REGION Network 10: Temperature Reached Conditions
   RUNG wire#powerrail
      Contact( #Selected )
      Contact( #Running )
      Contact( #Started )
      wire#w1
      { S7_Templates := "SrcType := Int" } EQ_Contact(in1 := #TemperatureControlSel, in2 := 0)
      wire#w2
      { S7_Templates := "SrcType := Real" } GE_Contact(in1 := #ActualTemperature, in2 := #SetTemperature)
      S_Coil( #HeatTempReached )
   END_RUNG
   RUNG wire#w2
      { S7_Templates := "SrcType := Real" } LE_Contact(in1 := #ActualTemperature, in2 := #TemperatureTolNeg)
      R_Coil( #HeatTempReached )
   END_RUNG
   RUNG wire#w1
      { S7_Templates := "SrcType := Int" } EQ_Contact(in1 := #TemperatureControlSel, in2 := 1)
      wire#w3
      { S7_Templates := "SrcType := Real" } LE_Contact(in1 := #ActualTemperature, in2 := #SetTemperature)
      S_Coil( #CoolTempReached )
   END_RUNG
   RUNG wire#w3
      { S7_Templates := "SrcType := Real" } GE_Contact(in1 := #ActualTemperature, in2 := #TemperatureTolPos)
      R_Coil( #CoolTempReached )
   END_RUNG
   // the same network as SCL:
   #_w1 := #Selected AND #Running AND #Started;
   #_w2 := #_w1 AND (#TemperatureControlSel = 0);
   IF #_w2 AND (#ActualTemperature >= #SetTemperature) THEN #HeatTempReached := TRUE; END_IF;
   IF #_w2 AND (#ActualTemperature <= #TemperatureTolNeg) THEN #HeatTempReached := FALSE; END_IF;
   #_w3 := #_w1 AND (#TemperatureControlSel = 1);
   IF #_w3 AND (#ActualTemperature <= #SetTemperature) THEN #CoolTempReached := TRUE; END_IF;
   IF #_w3 AND (#ActualTemperature >= #TemperatureTolPos) THEN #CoolTempReached := FALSE; END_IF;
END_REGION

REGION Network 11: Timer
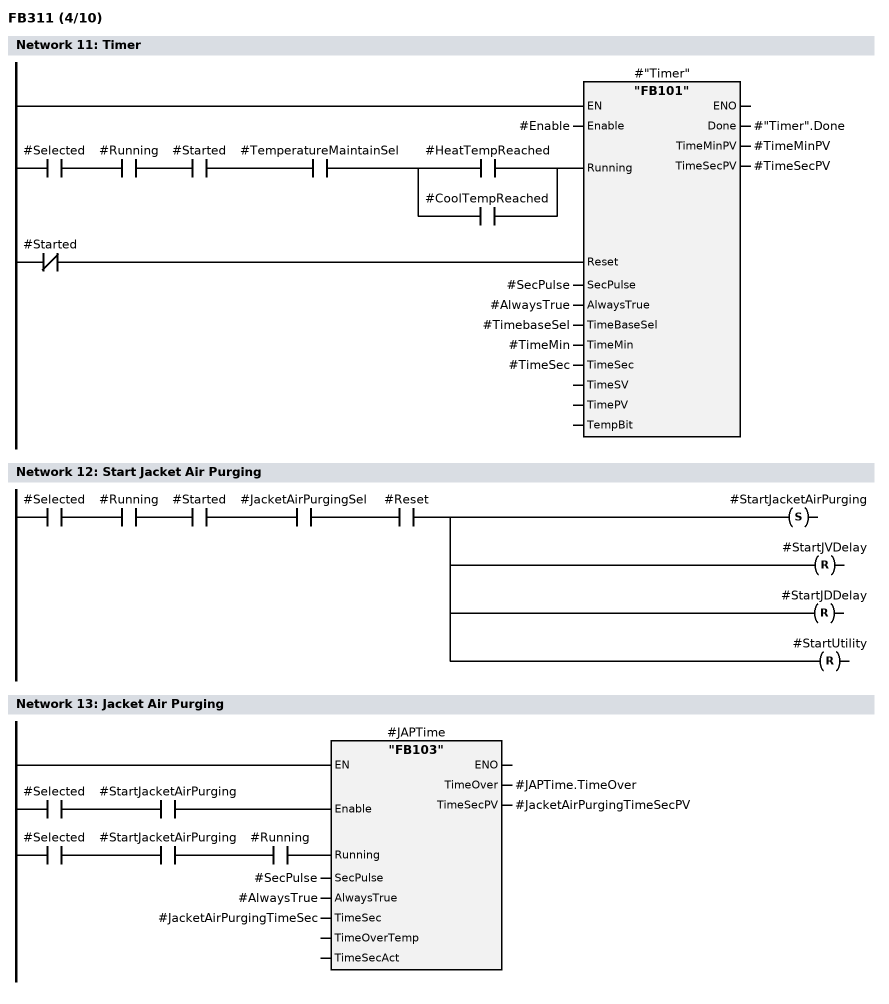
   RUNG wire#powerrail
      #"Timer"(Running := wire#w2, Reset := wire#w3, Enable := #Enable, SecPulse := #SecPulse, AlwaysTrue := #AlwaysTrue, TimeBaseSel := #TimebaseSel, TimeMin := #TimeMin, TimeSec := #TimeSec, TimeSV :=, TimePV :=, TempBit :=, Done => #"Timer".Done, TimeMinPV => #TimeMinPV, TimeSecPV => #TimeSecPV)
   END_RUNG
   RUNG wire#powerrail
      Contact( #Selected )
      Contact( #Running )
      Contact( #Started )
      Contact( #TemperatureMaintainSel )
      wire#w1
      Contact( #HeatTempReached )
   END_RUNG wire#w2
   RUNG wire#w1
      Contact( #CoolTempReached )
   END_RUNG wire#w2
   RUNG wire#powerrail
      I_Contact( #Started )
   END_RUNG wire#w3
   // the same network as SCL:
   #"Timer"(Enable := #Enable,   // "FB101"
            Running := #Selected AND #Running AND #Started AND #TemperatureMaintainSel AND (#HeatTempReached OR #CoolTempReached),
            Reset := NOT #Started,
            SecPulse := #SecPulse,
            AlwaysTrue := #AlwaysTrue,
            TimeBaseSel := #TimebaseSel,
            TimeMin := #TimeMin,
            TimeSec := #TimeSec,
            Done => #"Timer".Done,
            TimeMinPV => #TimeMinPV,
            TimeSecPV => #TimeSecPV);
END_REGION

REGION Network 12: Start Jacket Air Purging
   RUNG wire#powerrail
      Contact( #Selected )
      Contact( #Running )
      Contact( #Started )
      Contact( #JacketAirPurgingSel )
      Contact( #Reset )
      wire#w1
      S_Coil( #StartJacketAirPurging )
   END_RUNG
   RUNG wire#w1
      R_Coil( #StartJVDelay )
   END_RUNG
   RUNG wire#w1
      R_Coil( #StartJDDelay )
   END_RUNG
   RUNG wire#w1
      R_Coil( #StartUtility )
   END_RUNG
   // the same network as SCL:
   IF #Selected AND #Running AND #Started AND #JacketAirPurgingSel AND #Reset THEN
       #StartJacketAirPurging := TRUE;
       #StartJVDelay := FALSE;
       #StartJDDelay := FALSE;
       #StartUtility := FALSE;
   END_IF;
END_REGION

REGION Network 13: Jacket Air Purging
   RUNG wire#powerrail
      #JAPTime(Enable := wire#w1, Running := wire#w2, SecPulse := #SecPulse, AlwaysTrue := #AlwaysTrue, TimeSec := #JacketAirPurgingTimeSec, TimeOverTemp :=, TimeSecAct :=, TimeOver => #JAPTime.TimeOver, TimeSecPV => #JacketAirPurgingTimeSecPV)
   END_RUNG
   RUNG wire#powerrail
      Contact( #Selected )
      Contact( #StartJacketAirPurging )
   END_RUNG wire#w1
   RUNG wire#powerrail
      Contact( #Selected )
      Contact( #StartJacketAirPurging )
      Contact( #Running )
   END_RUNG wire#w2
   // the same network as SCL:
   #JAPTime(Enable := #Selected AND #StartJacketAirPurging,   // "FB103"
            Running := #Selected AND #StartJacketAirPurging AND #Running,
            SecPulse := #SecPulse,
            AlwaysTrue := #AlwaysTrue,
            TimeSec := #JacketAirPurgingTimeSec,
            TimeOver => #JAPTime.TimeOver,
            TimeSecPV => #JacketAirPurgingTimeSecPV);
END_REGION

REGION Network 14: Over
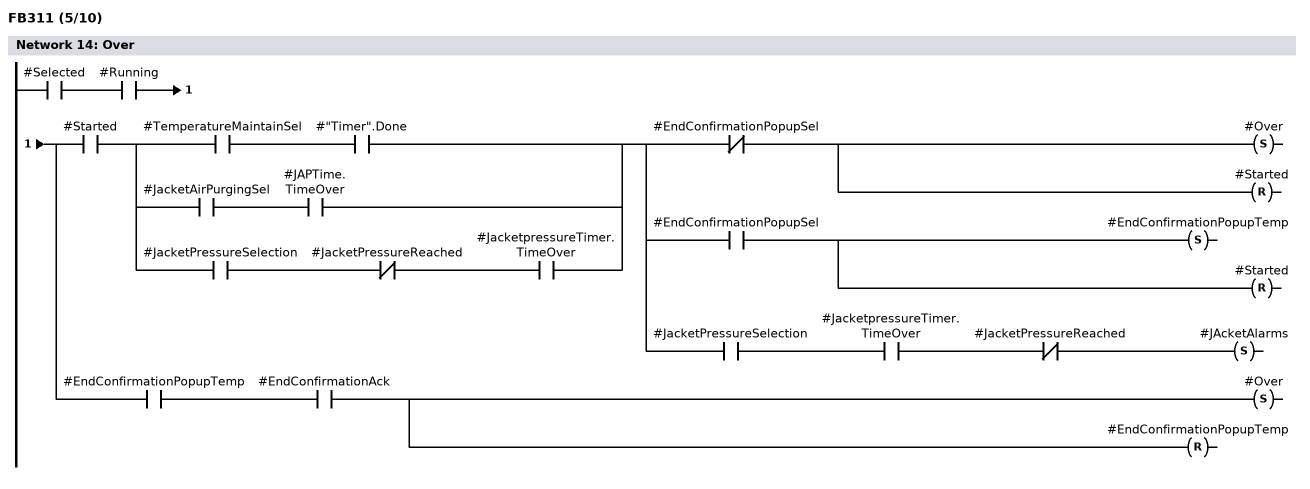
   RUNG wire#powerrail
      Contact( #Selected )
      Contact( #Running )
      wire#w1
      Contact( #Started )
      wire#w2
      Contact( #TemperatureMaintainSel )
      Contact( #"Timer".Done )
      wire#w3
      I_Contact( #EndConfirmationPopupSel )
      wire#w4
      S_Coil( #Over )
   END_RUNG
   RUNG wire#w2
      Contact( #JacketAirPurgingSel )
      Contact( #JAPTime.TimeOver )
   END_RUNG wire#w3
   RUNG wire#w2
      Contact( #JacketPressureSelection )
      I_Contact( #JacketPressureReached )
      Contact( #JacketpressureTimer.TimeOver )
   END_RUNG wire#w3
   RUNG wire#w4
      R_Coil( #Started )
   END_RUNG
   RUNG wire#w3
      Contact( #EndConfirmationPopupSel )
      wire#w5
      S_Coil( #EndConfirmationPopupTemp )
   END_RUNG
   RUNG wire#w5
      R_Coil( #Started )
   END_RUNG
   RUNG wire#w3
      Contact( #JacketPressureSelection )
      Contact( #JacketpressureTimer.TimeOver )
      I_Contact( #JacketPressureReached )
      S_Coil( #JAcketAlarms )
   END_RUNG
   RUNG wire#w1
      Contact( #EndConfirmationPopupTemp )
      Contact( #EndConfirmationAck )
      wire#w6
      S_Coil( #Over )
   END_RUNG
   RUNG wire#w6
      R_Coil( #EndConfirmationPopupTemp )
   END_RUNG
   // the same network as SCL:
   #_w1 := #Selected AND #Running;
   #_w2 := #_w1 AND #Started AND ((#TemperatureMaintainSel AND #"Timer".Done) OR (#JacketAirPurgingSel AND #JAPTime.TimeOver) OR (#JacketPressureSelection AND NOT #JacketPressureReached AND #JacketpressureTimer.TimeOver));
   IF #_w2 AND NOT #EndConfirmationPopupSel THEN
       #Over := TRUE;
       #Started := FALSE;
   END_IF;
   IF #_w2 AND #EndConfirmationPopupSel THEN
       #EndConfirmationPopupTemp := TRUE;
       #Started := FALSE;
   END_IF;
   IF #_w2 AND #JacketPressureSelection AND #JacketpressureTimer.TimeOver AND NOT #JacketPressureReached THEN
       #JAcketAlarms := TRUE;
   END_IF;
   IF #_w1 AND #EndConfirmationPopupTemp AND #EndConfirmationAck THEN
       #Over := TRUE;
       #EndConfirmationPopupTemp := FALSE;
   END_IF;
END_REGION

REGION Network 15: Outputs
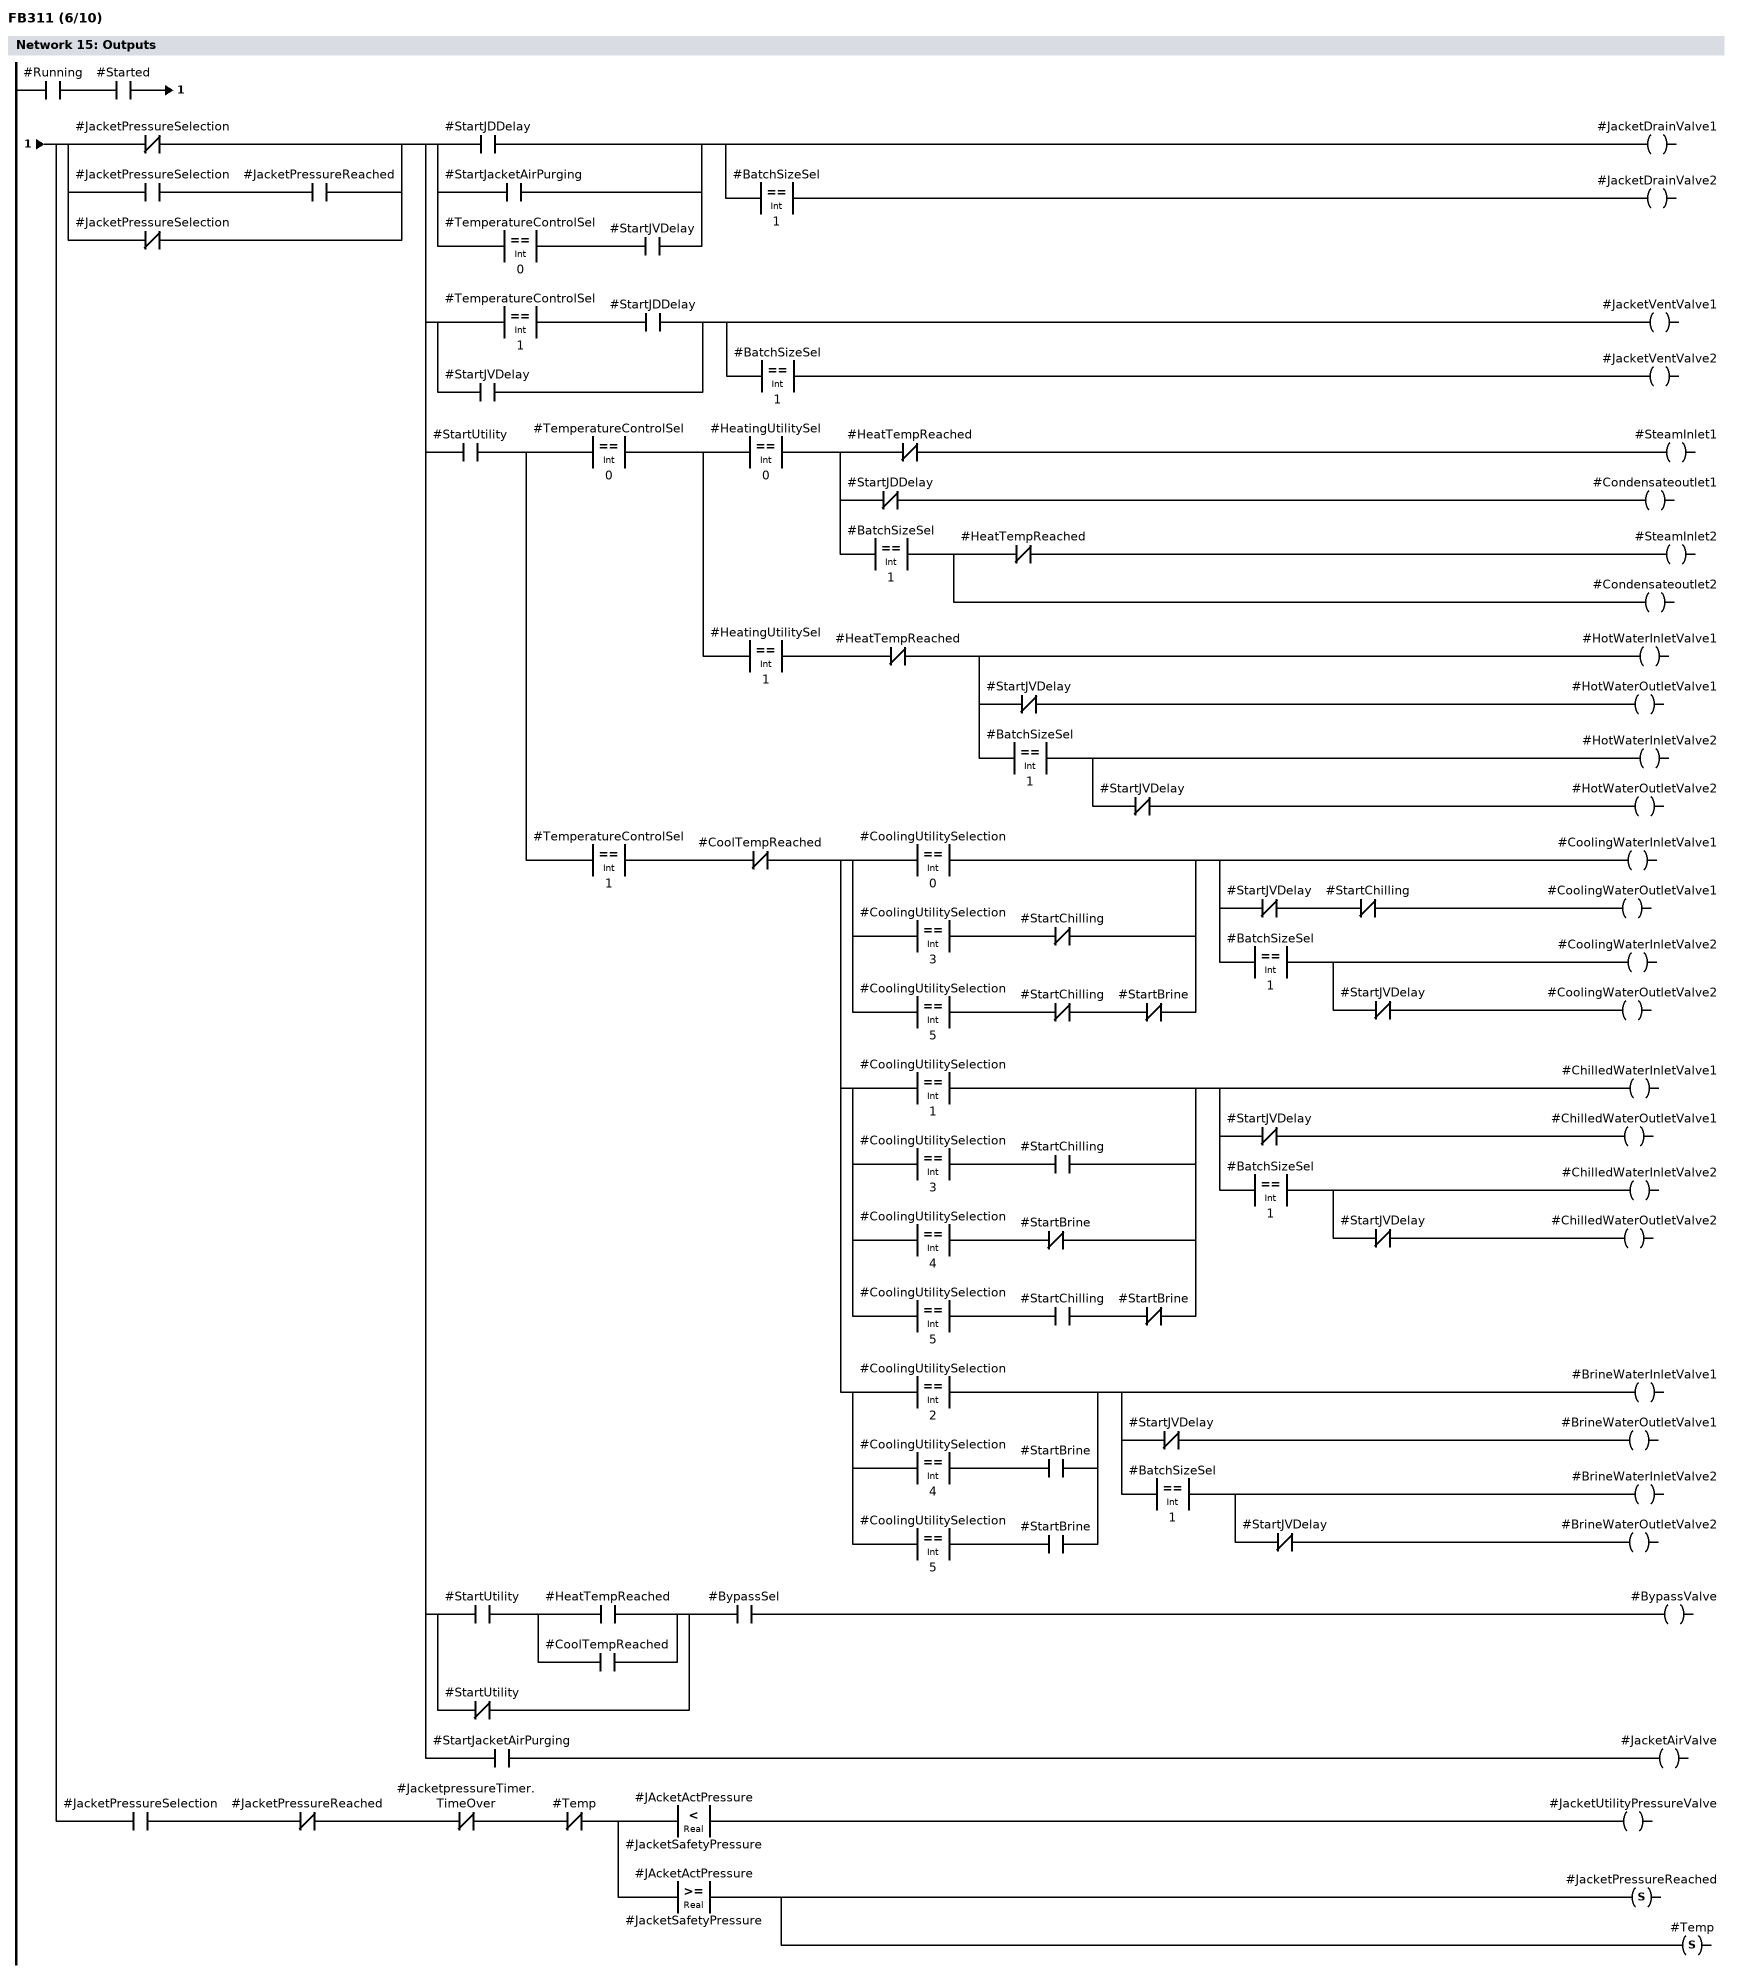
   RUNG wire#powerrail
      Contact( #Running )
      Contact( #Started )
      wire#w1
      I_Contact( #JacketPressureSelection )
      wire#w2
      Contact( #StartJDDelay )
      wire#w3
      Coil( #JacketDrainValve1 )
   END_RUNG
   RUNG wire#w1
      Contact( #JacketPressureSelection )
      Contact( #JacketPressureReached )
   END_RUNG wire#w2
   RUNG wire#w1
      I_Contact( #JacketPressureSelection )
   END_RUNG wire#w2
   RUNG wire#w2
      Contact( #StartJacketAirPurging )
   END_RUNG wire#w3
   RUNG wire#w2
      { S7_Templates := "SrcType := Int" } EQ_Contact(in1 := #TemperatureControlSel, in2 := 0)
      Contact( #StartJVDelay )
   END_RUNG wire#w3
   RUNG wire#w3
      { S7_Templates := "SrcType := Int" } EQ_Contact(in1 := #BatchSizeSel, in2 := 1)
      Coil( #JacketDrainValve2 )
   END_RUNG
   RUNG wire#w2
      { S7_Templates := "SrcType := Int" } EQ_Contact(in1 := #TemperatureControlSel, in2 := 1)
      Contact( #StartJDDelay )
      wire#w4
      Coil( #JacketVentValve1 )
   END_RUNG
   RUNG wire#w2
      Contact( #StartJVDelay )
   END_RUNG wire#w4
   RUNG wire#w4
      { S7_Templates := "SrcType := Int" } EQ_Contact(in1 := #BatchSizeSel, in2 := 1)
      Coil( #JacketVentValve2 )
   END_RUNG
   RUNG wire#w2
      Contact( #StartUtility )
      wire#w5
      { S7_Templates := "SrcType := Int" } EQ_Contact(in1 := #TemperatureControlSel, in2 := 0)
      wire#w6
      { S7_Templates := "SrcType := Int" } EQ_Contact(in1 := #HeatingUtilitySel, in2 := 0)
      wire#w7
      I_Contact( #HeatTempReached )
      Coil( #SteamInlet1 )
   END_RUNG
   RUNG wire#w7
      I_Contact( #StartJDDelay )
      Coil( #Condensateoutlet1 )
   END_RUNG
   RUNG wire#w7
      { S7_Templates := "SrcType := Int" } EQ_Contact(in1 := #BatchSizeSel, in2 := 1)
      wire#w8
      I_Contact( #HeatTempReached )
      Coil( #SteamInlet2 )
   END_RUNG
   RUNG wire#w8
      Coil( #Condensateoutlet2 )
   END_RUNG
   RUNG wire#w6
      { S7_Templates := "SrcType := Int" } EQ_Contact(in1 := #HeatingUtilitySel, in2 := 1)
      I_Contact( #HeatTempReached )
      wire#w9
      Coil( #HotWaterInletValve1 )
   END_RUNG
   RUNG wire#w9
      I_Contact( #StartJVDelay )
      Coil( #HotWaterOutletValve1 )
   END_RUNG
   RUNG wire#w9
      { S7_Templates := "SrcType := Int" } EQ_Contact(in1 := #BatchSizeSel, in2 := 1)
      wire#w10
      Coil( #HotWaterInletValve2 )
   END_RUNG
   RUNG wire#w10
      I_Contact( #StartJVDelay )
      Coil( #HotWaterOutletValve2 )
   END_RUNG
   RUNG wire#w5
      { S7_Templates := "SrcType := Int" } EQ_Contact(in1 := #TemperatureControlSel, in2 := 1)
      I_Contact( #CoolTempReached )
      wire#w11
      { S7_Templates := "SrcType := Int" } EQ_Contact(in1 := #CoolingUtilitySelection, in2 := 0)
      wire#w12
      Coil( #CoolingWaterInletValve1 )
   END_RUNG
   RUNG wire#w11
      { S7_Templates := "SrcType := Int" } EQ_Contact(in1 := #CoolingUtilitySelection, in2 := 3)
      I_Contact( #StartChilling )
   END_RUNG wire#w12
   RUNG wire#w11
      { S7_Templates := "SrcType := Int" } EQ_Contact(in1 := #CoolingUtilitySelection, in2 := 5)
      I_Contact( #StartChilling )
      I_Contact( #StartBrine )
   END_RUNG wire#w12
   RUNG wire#w12
      I_Contact( #StartJVDelay )
      I_Contact( #StartChilling )
      Coil( #CoolingWaterOutletValve1 )
   END_RUNG
   RUNG wire#w12
      { S7_Templates := "SrcType := Int" } EQ_Contact(in1 := #BatchSizeSel, in2 := 1)
      wire#w13
      Coil( #CoolingWaterInletValve2 )
   END_RUNG
   RUNG wire#w13
      I_Contact( #StartJVDelay )
      Coil( #CoolingWaterOutletValve2 )
   END_RUNG
   RUNG wire#w11
      { S7_Templates := "SrcType := Int" } EQ_Contact(in1 := #CoolingUtilitySelection, in2 := 1)
      wire#w14
      Coil( #ChilledWaterInletValve1 )
   END_RUNG
   RUNG wire#w11
      { S7_Templates := "SrcType := Int" } EQ_Contact(in1 := #CoolingUtilitySelection, in2 := 3)
      Contact( #StartChilling )
   END_RUNG wire#w14
   RUNG wire#w11
      { S7_Templates := "SrcType := Int" } EQ_Contact(in1 := #CoolingUtilitySelection, in2 := 4)
      I_Contact( #StartBrine )
   END_RUNG wire#w14
   RUNG wire#w11
      { S7_Templates := "SrcType := Int" } EQ_Contact(in1 := #CoolingUtilitySelection, in2 := 5)
      Contact( #StartChilling )
      I_Contact( #StartBrine )
   END_RUNG wire#w14
   RUNG wire#w14
      I_Contact( #StartJVDelay )
      Coil( #ChilledWaterOutletValve1 )
   END_RUNG
   RUNG wire#w14
      { S7_Templates := "SrcType := Int" } EQ_Contact(in1 := #BatchSizeSel, in2 := 1)
      wire#w15
      Coil( #ChilledWaterInletValve2 )
   END_RUNG
   RUNG wire#w15
      I_Contact( #StartJVDelay )
      Coil( #ChilledWaterOutletValve2 )
   END_RUNG
   RUNG wire#w11
      { S7_Templates := "SrcType := Int" } EQ_Contact(in1 := #CoolingUtilitySelection, in2 := 2)
      wire#w16
      Coil( #BrineWaterInletValve1 )
   END_RUNG
   RUNG wire#w11
      { S7_Templates := "SrcType := Int" } EQ_Contact(in1 := #CoolingUtilitySelection, in2 := 4)
      Contact( #StartBrine )
   END_RUNG wire#w16
   RUNG wire#w11
      { S7_Templates := "SrcType := Int" } EQ_Contact(in1 := #CoolingUtilitySelection, in2 := 5)
      Contact( #StartBrine )
   END_RUNG wire#w16
   RUNG wire#w16
      I_Contact( #StartJVDelay )
      Coil( #BrineWaterOutletValve1 )
   END_RUNG
   RUNG wire#w16
      { S7_Templates := "SrcType := Int" } EQ_Contact(in1 := #BatchSizeSel, in2 := 1)
      wire#w17
      Coil( #BrineWaterInletValve2 )
   END_RUNG
   RUNG wire#w17
      I_Contact( #StartJVDelay )
      Coil( #BrineWaterOutletValve2 )
   END_RUNG
   RUNG wire#w2
      Contact( #StartUtility )
      wire#w18
      Contact( #HeatTempReached )
      wire#w19
      Contact( #BypassSel )
      Coil( #BypassValve )
   END_RUNG
   RUNG wire#w18
      Contact( #CoolTempReached )
   END_RUNG wire#w19
   RUNG wire#w2
      I_Contact( #StartUtility )
   END_RUNG wire#w19
   RUNG wire#w2
      Contact( #StartJacketAirPurging )
      Coil( #JacketAirValve )
   END_RUNG
   RUNG wire#w1
      Contact( #JacketPressureSelection )
      I_Contact( #JacketPressureReached )
      I_Contact( #JacketpressureTimer.TimeOver )
      I_Contact( #Temp )
      wire#w20
      { S7_Templates := "SrcType := Real" } LT_Contact(in1 := #JAcketActPressure, in2 := #JacketSafetyPressure)
      Coil( #JacketUtilityPressureValve )
   END_RUNG
   RUNG wire#w20
      { S7_Templates := "SrcType := Real" } GE_Contact(in1 := #JAcketActPressure, in2 := #JacketSafetyPressure)
      wire#w21
      S_Coil( #JacketPressureReached )
   END_RUNG
   RUNG wire#w21
      S_Coil( #Temp )
   END_RUNG
   // the same network as SCL:
   #_w1 := #Running AND #Started;
   #_w2 := #_w1 AND (NOT #JacketPressureSelection OR (#JacketPressureSelection AND #JacketPressureReached) OR NOT #JacketPressureSelection);
   #JacketDrainValve1 := #_w2 AND (#StartJDDelay OR #StartJacketAirPurging OR ((#TemperatureControlSel = 0) AND #StartJVDelay));
   #JacketDrainValve2 := #JacketDrainValve1 AND (#BatchSizeSel = 1);
   #JacketVentValve1 := #_w2 AND (((#TemperatureControlSel = 1) AND #StartJDDelay) OR #StartJVDelay);
   #JacketVentValve2 := #JacketVentValve1 AND (#BatchSizeSel = 1);
   #_w3 := #_w2 AND #StartUtility;
   #_w4 := #_w3 AND (#TemperatureControlSel = 0);
   #_w5 := #_w4 AND (#HeatingUtilitySel = 0);
   #SteamInlet1 := #_w5 AND NOT #HeatTempReached;
   #Condensateoutlet1 := #_w5 AND NOT #StartJDDelay;
   #_w6 := #_w5 AND (#BatchSizeSel = 1);
   #SteamInlet2 := #_w6 AND NOT #HeatTempReached;
   #Condensateoutlet2 := #_w6;
   #HotWaterInletValve1 := #_w4 AND (#HeatingUtilitySel = 1) AND NOT #HeatTempReached;
   #HotWaterOutletValve1 := #HotWaterInletValve1 AND NOT #StartJVDelay;
   #HotWaterInletValve2 := #HotWaterInletValve1 AND (#BatchSizeSel = 1);
   #HotWaterOutletValve2 := #HotWaterInletValve2 AND NOT #StartJVDelay;
   #_w7 := #_w3 AND (#TemperatureControlSel = 1) AND NOT #CoolTempReached;
   #CoolingWaterInletValve1 := #_w7 AND ((#CoolingUtilitySelection = 0) OR ((#CoolingUtilitySelection = 3) AND NOT #StartChilling) OR ((#CoolingUtilitySelection = 5) AND NOT #StartChilling AND NOT #StartBrine));
   #CoolingWaterOutletValve1 := #CoolingWaterInletValve1 AND NOT #StartJVDelay AND NOT #StartChilling;
   #CoolingWaterInletValve2 := #CoolingWaterInletValve1 AND (#BatchSizeSel = 1);
   #CoolingWaterOutletValve2 := #CoolingWaterInletValve2 AND NOT #StartJVDelay;
   #ChilledWaterInletValve1 := #_w7 AND ((#CoolingUtilitySelection = 1) OR ((#CoolingUtilitySelection = 3) AND #StartChilling) OR ((#CoolingUtilitySelection = 4) AND NOT #StartBrine) OR ((#CoolingUtilitySelection = 5) AND #StartChilling AND NOT #StartBrine));
   #ChilledWaterOutletValve1 := #ChilledWaterInletValve1 AND NOT #StartJVDelay;
   #ChilledWaterInletValve2 := #ChilledWaterInletValve1 AND (#BatchSizeSel = 1);
   #ChilledWaterOutletValve2 := #ChilledWaterInletValve2 AND NOT #StartJVDelay;
   #BrineWaterInletValve1 := #_w7 AND ((#CoolingUtilitySelection = 2) OR ((#CoolingUtilitySelection = 4) AND #StartBrine) OR ((#CoolingUtilitySelection = 5) AND #StartBrine));
   #BrineWaterOutletValve1 := #BrineWaterInletValve1 AND NOT #StartJVDelay;
   #BrineWaterInletValve2 := #BrineWaterInletValve1 AND (#BatchSizeSel = 1);
   #BrineWaterOutletValve2 := #BrineWaterInletValve2 AND NOT #StartJVDelay;
   #BypassValve := #_w2 AND ((#StartUtility AND (#HeatTempReached OR #CoolTempReached)) OR NOT #StartUtility) AND #BypassSel;
   #JacketAirValve := #_w2 AND #StartJacketAirPurging;
   #_w8 := #_w1 AND #JacketPressureSelection AND NOT #JacketPressureReached AND NOT #JacketpressureTimer.TimeOver AND NOT #Temp;
   #JacketUtilityPressureValve := #_w8 AND (#JAcketActPressure < #JacketSafetyPressure);
   IF #_w8 AND (#JAcketActPressure >= #JacketSafetyPressure) THEN
       #JacketPressureReached := TRUE;
       #Temp := TRUE;
   END_IF;
END_REGION

REGION Network 16: Jacket Air Purging
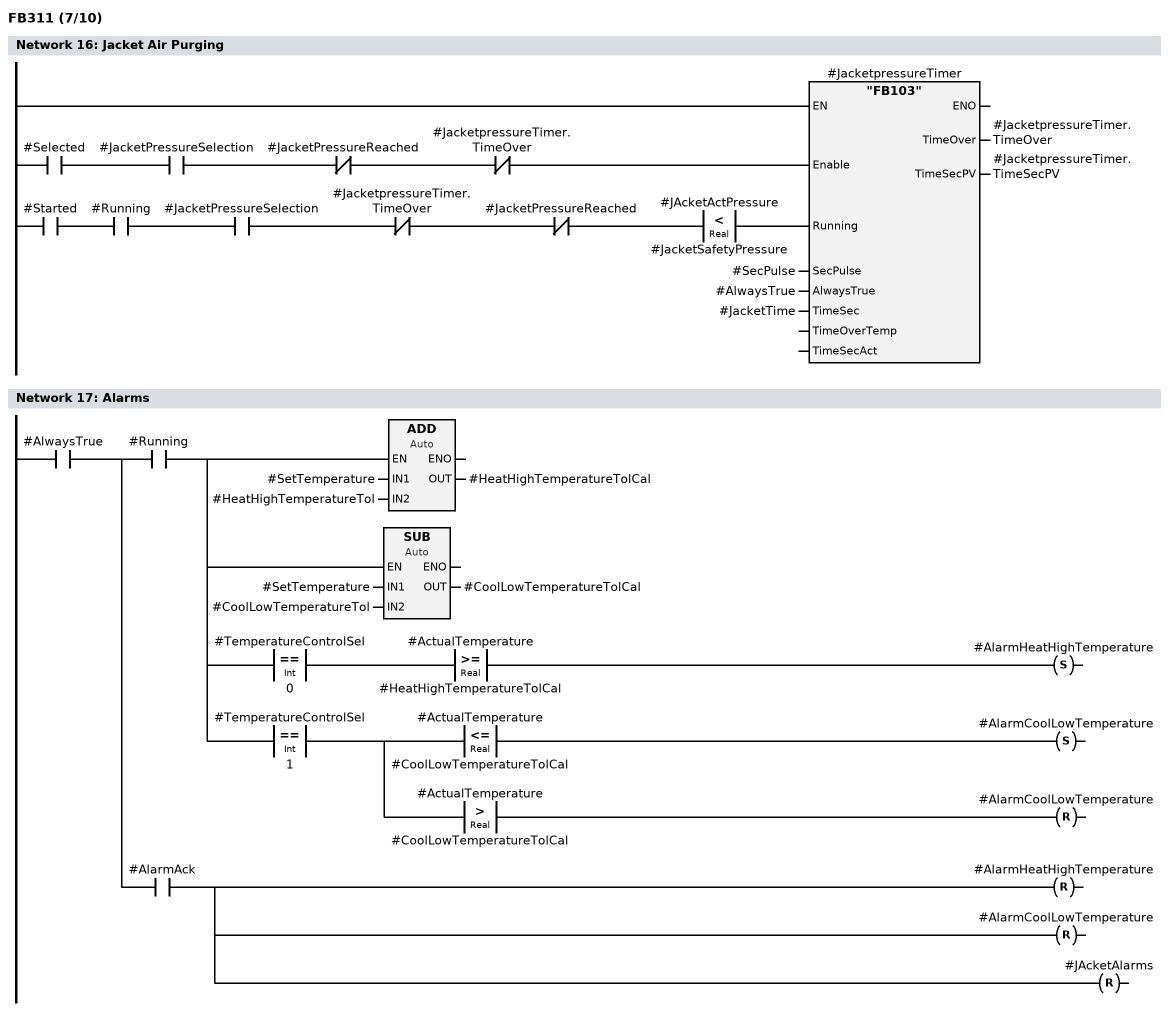
   RUNG wire#powerrail
      #JacketpressureTimer(Enable := wire#w1, Running := wire#w2, SecPulse := #SecPulse, AlwaysTrue := #AlwaysTrue, TimeSec := #JacketTime, TimeOverTemp :=, TimeSecAct :=, TimeOver => #JacketpressureTimer.TimeOver, TimeSecPV => #JacketpressureTimer.TimeSecPV)
   END_RUNG
   RUNG wire#powerrail
      Contact( #Selected )
      Contact( #JacketPressureSelection )
      I_Contact( #JacketPressureReached )
      I_Contact( #JacketpressureTimer.TimeOver )
   END_RUNG wire#w1
   RUNG wire#powerrail
      Contact( #Started )
      Contact( #Running )
      Contact( #JacketPressureSelection )
      I_Contact( #JacketpressureTimer.TimeOver )
      I_Contact( #JacketPressureReached )
      { S7_Templates := "SrcType := Real" } LT_Contact(in1 := #JAcketActPressure, in2 := #JacketSafetyPressure)
   END_RUNG wire#w2
   // the same network as SCL:
   #JacketpressureTimer(Enable := #Selected AND #JacketPressureSelection AND NOT #JacketPressureReached AND NOT #JacketpressureTimer.TimeOver,   // "FB103"
                        Running := #Started AND #Running AND #JacketPressureSelection AND NOT #JacketpressureTimer.TimeOver AND NOT #JacketPressureReached AND (#JAcketActPressure < #JacketSafetyPressure),
                        SecPulse := #SecPulse,
                        AlwaysTrue := #AlwaysTrue,
                        TimeSec := #JacketTime,
                        TimeOver => #JacketpressureTimer.TimeOver,
                        TimeSecPV => #JacketpressureTimer.TimeSecPV);
END_REGION

REGION Network 17: Alarms
   RUNG wire#powerrail
      Contact( #AlwaysTrue )
      wire#w1
      Contact( #Running )
      wire#w2
      Add(in1 := #SetTemperature, in2 := #HeatHighTemperatureTol, out => #HeatHighTemperatureTolCal)
   END_RUNG
   RUNG wire#w2
      Sub(in1 := #SetTemperature, in2 := #CoolLowTemperatureTol, out => #CoolLowTemperatureTolCal)
   END_RUNG
   RUNG wire#w2
      { S7_Templates := "SrcType := Int" } EQ_Contact(in1 := #TemperatureControlSel, in2 := 0)
      { S7_Templates := "SrcType := Real" } GE_Contact(in1 := #ActualTemperature, in2 := #HeatHighTemperatureTolCal)
      S_Coil( #AlarmHeatHighTemperature )
   END_RUNG
   RUNG wire#w2
      { S7_Templates := "SrcType := Int" } EQ_Contact(in1 := #TemperatureControlSel, in2 := 1)
      wire#w3
      { S7_Templates := "SrcType := Real" } LE_Contact(in1 := #ActualTemperature, in2 := #CoolLowTemperatureTolCal)
      S_Coil( #AlarmCoolLowTemperature )
   END_RUNG
   RUNG wire#w3
      { S7_Templates := "SrcType := Real" } GT_Contact(in1 := #ActualTemperature, in2 := #CoolLowTemperatureTolCal)
      R_Coil( #AlarmCoolLowTemperature )
   END_RUNG
   RUNG wire#w1
      Contact( #AlarmAck )
      wire#w4
      R_Coil( #AlarmHeatHighTemperature )
   END_RUNG
   RUNG wire#w4
      R_Coil( #AlarmCoolLowTemperature )
   END_RUNG
   RUNG wire#w4
      R_Coil( #JAcketAlarms )
   END_RUNG
   // the same network as SCL:
   #_w1 := #AlwaysTrue AND #Running;
   IF #_w1 THEN
       #HeatHighTemperatureTolCal := #SetTemperature + #HeatHighTemperatureTol;
       #CoolLowTemperatureTolCal := #SetTemperature - #CoolLowTemperatureTol;
   END_IF;
   IF #_w1 AND (#TemperatureControlSel = 0) AND (#ActualTemperature >= #HeatHighTemperatureTolCal) THEN
       #AlarmHeatHighTemperature := TRUE;
   END_IF;
   #_w2 := #_w1 AND (#TemperatureControlSel = 1);
   IF #_w2 AND (#ActualTemperature <= #CoolLowTemperatureTolCal) THEN
       #AlarmCoolLowTemperature := TRUE;
   END_IF;
   IF #_w2 AND (#ActualTemperature > #CoolLowTemperatureTolCal) THEN
       #AlarmCoolLowTemperature := FALSE;
   END_IF;
   IF #AlwaysTrue AND #AlarmAck THEN
       #AlarmHeatHighTemperature := FALSE;
       #AlarmCoolLowTemperature := FALSE;
       #JAcketAlarms := FALSE;
   END_IF;
END_REGION

REGION Network 18: Event Status
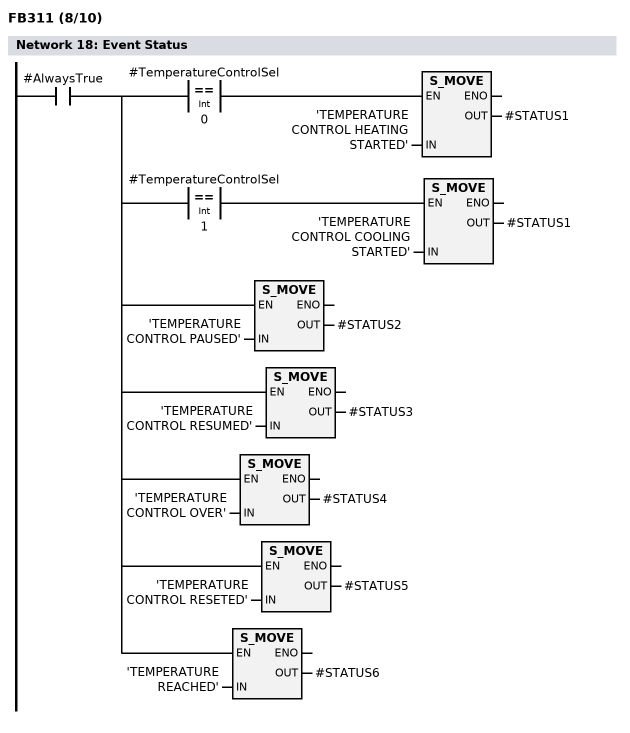
   RUNG wire#powerrail
      Contact( #AlwaysTrue )
      wire#w1
      { S7_Templates := "SrcType := Int" } EQ_Contact(in1 := #TemperatureControlSel, in2 := 0)
      S_Move(in := 'TEMPERATURE CONTROL HEATING STARTED', out => #STATUS1)
   END_RUNG
   RUNG wire#w1
      { S7_Templates := "SrcType := Int" } EQ_Contact(in1 := #TemperatureControlSel, in2 := 1)
      S_Move(in := 'TEMPERATURE CONTROL COOLING STARTED', out => #STATUS1)
   END_RUNG
   RUNG wire#w1
      S_Move(in := 'TEMPERATURE CONTROL PAUSED', out => #STATUS2)
   END_RUNG
   RUNG wire#w1
      S_Move(in := 'TEMPERATURE CONTROL RESUMED', out => #STATUS3)
   END_RUNG
   RUNG wire#w1
      S_Move(in := 'TEMPERATURE CONTROL OVER', out => #STATUS4)
   END_RUNG
   RUNG wire#w1
      S_Move(in := 'TEMPERATURE CONTROL RESETED', out => #STATUS5)
   END_RUNG
   RUNG wire#w1
      S_Move(in := 'TEMPERATURE REACHED', out => #STATUS6)
   END_RUNG
   // the same network as SCL:
   IF #AlwaysTrue AND (#TemperatureControlSel = 0) THEN
       #STATUS1 := 'TEMPERATURE CONTROL HEATING STARTED';
   END_IF;
   IF #AlwaysTrue AND (#TemperatureControlSel = 1) THEN
       #STATUS1 := 'TEMPERATURE CONTROL COOLING STARTED';
   END_IF;
   IF #AlwaysTrue THEN
       #STATUS2 := 'TEMPERATURE CONTROL PAUSED';
       #STATUS3 := 'TEMPERATURE CONTROL RESUMED';
       #STATUS4 := 'TEMPERATURE CONTROL OVER';
       #STATUS5 := 'TEMPERATURE CONTROL RESETED';
       #STATUS6 := 'TEMPERATURE REACHED';
   END_IF;
END_REGION

REGION Network 19: Print Logic
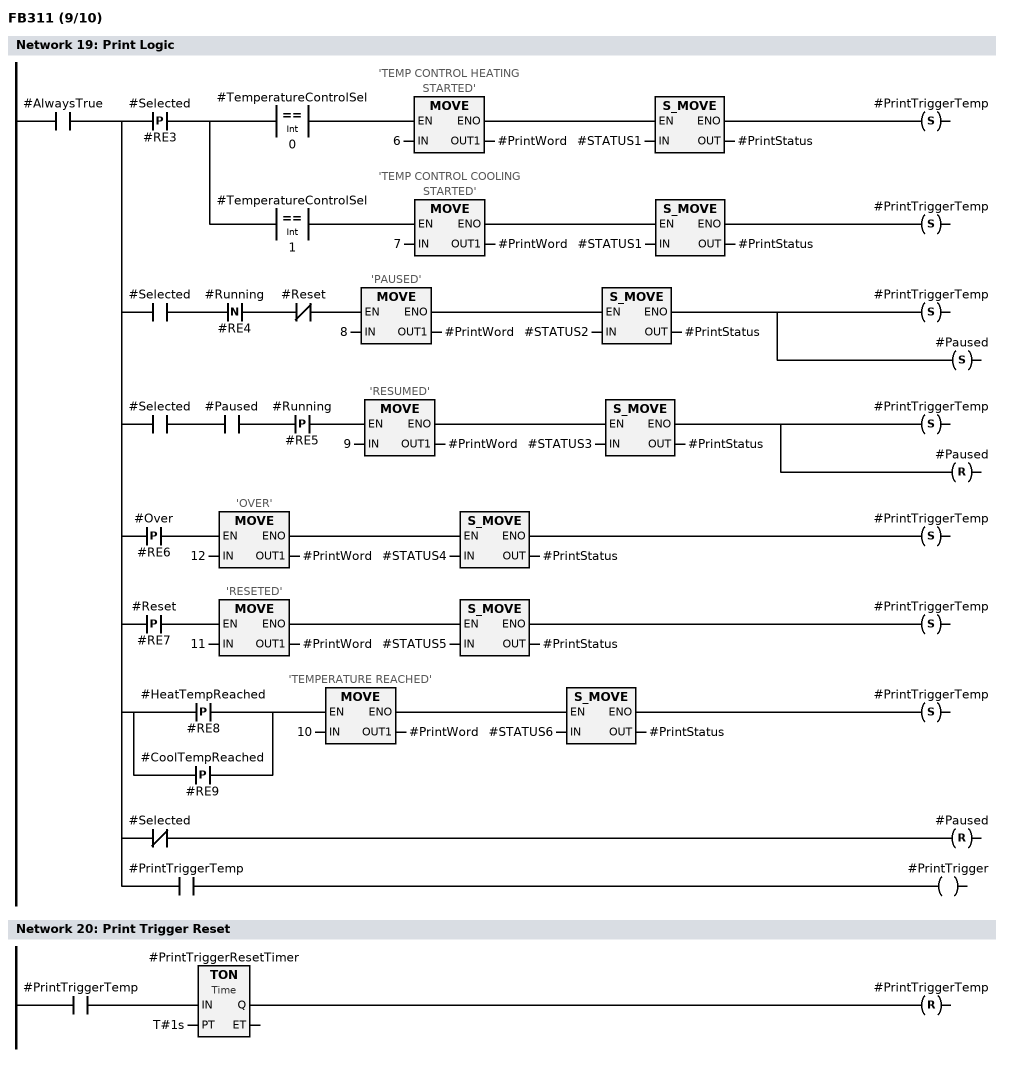
   RUNG wire#powerrail
      Contact( #AlwaysTrue )
      wire#w1
      P_Contact(operand := #Selected, bit := #RE3)
      wire#w2
      { S7_Templates := "SrcType := Int" } EQ_Contact(in1 := #TemperatureControlSel, in2 := 0)
      { S7_GenerateENO := "TRUE" } Move(in := 6, out1 => #PrintWord)   // 'TEMP CONTROL HEATING STARTED'
      S_Move(in := #STATUS1, out => #PrintStatus)
      S_Coil( #PrintTriggerTemp )
   END_RUNG
   RUNG wire#w2
      { S7_Templates := "SrcType := Int" } EQ_Contact(in1 := #TemperatureControlSel, in2 := 1)
      { S7_GenerateENO := "TRUE" } Move(in := 7, out1 => #PrintWord)   // 'TEMP CONTROL COOLING STARTED'
      S_Move(in := #STATUS1, out => #PrintStatus)
      S_Coil( #PrintTriggerTemp )
   END_RUNG
   RUNG wire#w1
      Contact( #Selected )
      N_Contact(operand := #Running, bit := #RE4)
      I_Contact( #Reset )
      { S7_GenerateENO := "TRUE" } Move(in := 8, out1 => #PrintWord)   // 'PAUSED'
      S_Move(in := #STATUS2, out => #PrintStatus)
      wire#w3
      S_Coil( #PrintTriggerTemp )
   END_RUNG
   RUNG wire#w3
      S_Coil( #Paused )
   END_RUNG
   RUNG wire#w1
      Contact( #Selected )
      Contact( #Paused )
      P_Contact(operand := #Running, bit := #RE5)
      { S7_GenerateENO := "TRUE" } Move(in := 9, out1 => #PrintWord)   // 'RESUMED'
      S_Move(in := #STATUS3, out => #PrintStatus)
      wire#w4
      S_Coil( #PrintTriggerTemp )
   END_RUNG
   RUNG wire#w4
      R_Coil( #Paused )
   END_RUNG
   RUNG wire#w1
      P_Contact(operand := #Over, bit := #RE6)
      { S7_GenerateENO := "TRUE" } Move(in := 12, out1 => #PrintWord)   // 'OVER'
      S_Move(in := #STATUS4, out => #PrintStatus)
      S_Coil( #PrintTriggerTemp )
   END_RUNG
   RUNG wire#w1
      P_Contact(operand := #Reset, bit := #RE7)
      { S7_GenerateENO := "TRUE" } Move(in := 11, out1 => #PrintWord)   // 'RESETED'
      S_Move(in := #STATUS5, out => #PrintStatus)
      S_Coil( #PrintTriggerTemp )
   END_RUNG
   RUNG wire#w1
      P_Contact(operand := #HeatTempReached, bit := #RE8)
      wire#w5
      { S7_GenerateENO := "TRUE" } Move(in := 10, out1 => #PrintWord)   // 'TEMPERATURE REACHED'
      S_Move(in := #STATUS6, out => #PrintStatus)
      S_Coil( #PrintTriggerTemp )
   END_RUNG
   RUNG wire#w1
      P_Contact(operand := #CoolTempReached, bit := #RE9)
   END_RUNG wire#w5
   RUNG wire#w1
      I_Contact( #Selected )
      R_Coil( #Paused )
   END_RUNG
   RUNG wire#w1
      Contact( #PrintTriggerTemp )
      Coil( #PrintTrigger )
   END_RUNG
   // the same network as SCL:
   // ENO of a box is taken as its EN; it also drops when the box reports an error
   #_w1 := #AlwaysTrue AND #Selected AND NOT #RE3;   // rising edge of #Selected
   #RE3 := #Selected;
   IF #_w1 AND (#TemperatureControlSel = 0) THEN
       #PrintWord := 6;   // 'TEMP CONTROL HEATING STARTED'
       #PrintStatus := #STATUS1;
       #PrintTriggerTemp := TRUE;
   END_IF;
   IF #_w1 AND (#TemperatureControlSel = 1) THEN
       #PrintWord := 7;   // 'TEMP CONTROL COOLING STARTED'
       #PrintStatus := #STATUS1;
       #PrintTriggerTemp := TRUE;
   END_IF;
   #_w2 := #AlwaysTrue AND #Selected AND NOT #Running AND #RE4;   // falling edge of #Running
   #RE4 := #Running;
   IF #_w2 AND NOT #Reset THEN
       #PrintWord := 8;   // 'PAUSED'
       #PrintStatus := #STATUS2;
       #PrintTriggerTemp := TRUE;
       #Paused := TRUE;
   END_IF;
   #_w3 := #AlwaysTrue AND #Selected AND #Paused AND #Running AND NOT #RE5;   // rising edge of #Running
   #RE5 := #Running;
   IF #_w3 THEN
       #PrintWord := 9;   // 'RESUMED'
       #PrintStatus := #STATUS3;
       #PrintTriggerTemp := TRUE;
       #Paused := FALSE;
   END_IF;
   #_w4 := #AlwaysTrue AND #Over AND NOT #RE6;   // rising edge of #Over
   #RE6 := #Over;
   IF #_w4 THEN
       #PrintWord := 12;   // 'OVER'
       #PrintStatus := #STATUS4;
       #PrintTriggerTemp := TRUE;
   END_IF;
   #_w5 := #AlwaysTrue AND #Reset AND NOT #RE7;   // rising edge of #Reset
   #RE7 := #Reset;
   IF #_w5 THEN
       #PrintWord := 11;   // 'RESETED'
       #PrintStatus := #STATUS5;
       #PrintTriggerTemp := TRUE;
   END_IF;
   #_w6 := #AlwaysTrue AND #HeatTempReached AND NOT #RE8;   // rising edge of #HeatTempReached
   #RE8 := #HeatTempReached;
   #_w7 := #AlwaysTrue AND #CoolTempReached AND NOT #RE9;   // rising edge of #CoolTempReached
   #RE9 := #CoolTempReached;
   IF #_w6 OR #_w7 THEN
       #PrintWord := 10;   // 'TEMPERATURE REACHED'
       #PrintStatus := #STATUS6;
       #PrintTriggerTemp := TRUE;
   END_IF;
   IF #AlwaysTrue AND NOT #Selected THEN #Paused := FALSE; END_IF;
   #PrintTrigger := #AlwaysTrue AND #PrintTriggerTemp;
END_REGION

REGION Network 20: Print Trigger Reset
   RUNG wire#powerrail
      Contact( #PrintTriggerTemp )
      { S7_Templates := "time_type := Time" } #PrintTriggerResetTimer.TON(pt := T#1s, et =>)
      R_Coil( #PrintTriggerTemp )
   END_RUNG
   // the same network as SCL:
   #PrintTriggerResetTimer(IN := #PrintTriggerTemp, PT := T#1s);   // TON
   IF #PrintTriggerResetTimer.Q THEN #PrintTriggerTemp := FALSE; END_IF;
END_REGION

REGION Network 21: Button Reset
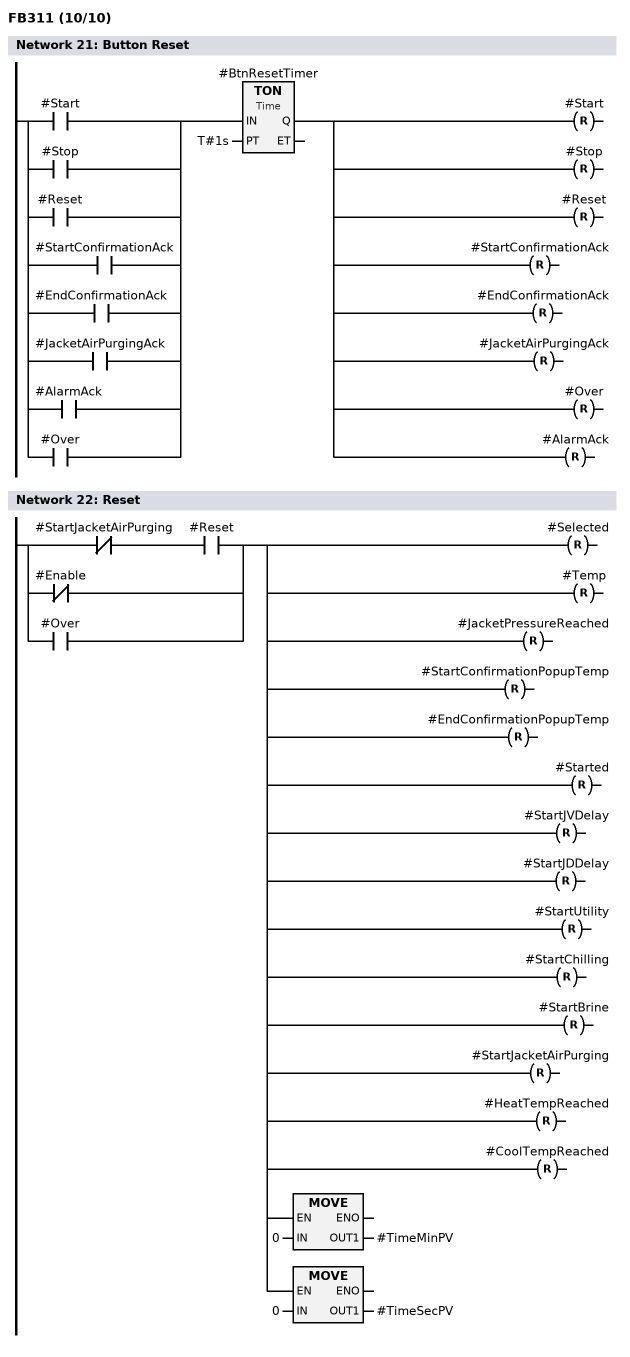
   RUNG wire#powerrail
      Contact( #Start )
      wire#w1
      { S7_Templates := "time_type := Time" } #BtnResetTimer.TON(pt := T#1s, et =>)
      wire#w2
      R_Coil( #Start )
   END_RUNG
   RUNG wire#powerrail
      Contact( #Stop )
   END_RUNG wire#w1
   RUNG wire#powerrail
      Contact( #Reset )
   END_RUNG wire#w1
   RUNG wire#powerrail
      Contact( #StartConfirmationAck )
   END_RUNG wire#w1
   RUNG wire#powerrail
      Contact( #EndConfirmationAck )
   END_RUNG wire#w1
   RUNG wire#powerrail
      Contact( #JacketAirPurgingAck )
   END_RUNG wire#w1
   RUNG wire#powerrail
      Contact( #AlarmAck )
   END_RUNG wire#w1
   RUNG wire#powerrail
      Contact( #Over )
   END_RUNG wire#w1
   RUNG wire#w2
      R_Coil( #Stop )
   END_RUNG
   RUNG wire#w2
      R_Coil( #Reset )
   END_RUNG
   RUNG wire#w2
      R_Coil( #StartConfirmationAck )
   END_RUNG
   RUNG wire#w2
      R_Coil( #EndConfirmationAck )
   END_RUNG
   RUNG wire#w2
      R_Coil( #JacketAirPurgingAck )
   END_RUNG
   RUNG wire#w2
      R_Coil( #Over )
   END_RUNG
   RUNG wire#w2
      R_Coil( #AlarmAck )
   END_RUNG
   // the same network as SCL:
   #BtnResetTimer(IN := #Start OR #Stop OR #Reset OR #StartConfirmationAck OR #EndConfirmationAck OR #JacketAirPurgingAck OR #AlarmAck OR #Over,   // TON
                  PT := T#1s);
   IF #BtnResetTimer.Q THEN
       #Start := FALSE;
       #Stop := FALSE;
       #Reset := FALSE;
       #StartConfirmationAck := FALSE;
       #EndConfirmationAck := FALSE;
       #JacketAirPurgingAck := FALSE;
       #Over := FALSE;
       #AlarmAck := FALSE;
   END_IF;
END_REGION

REGION Network 22: Reset
   RUNG wire#powerrail
      I_Contact( #StartJacketAirPurging )
      Contact( #Reset )
      wire#w1
      R_Coil( #Selected )
   END_RUNG
   RUNG wire#powerrail
      I_Contact( #Enable )
   END_RUNG wire#w1
   RUNG wire#powerrail
      Contact( #Over )
   END_RUNG wire#w1
   RUNG wire#w1
      R_Coil( #Temp )
   END_RUNG
   RUNG wire#w1
      R_Coil( #JacketPressureReached )
   END_RUNG
   RUNG wire#w1
      R_Coil( #StartConfirmationPopupTemp )
   END_RUNG
   RUNG wire#w1
      R_Coil( #EndConfirmationPopupTemp )
   END_RUNG
   RUNG wire#w1
      R_Coil( #Started )
   END_RUNG
   RUNG wire#w1
      R_Coil( #StartJVDelay )
   END_RUNG
   RUNG wire#w1
      R_Coil( #StartJDDelay )
   END_RUNG
   RUNG wire#w1
      R_Coil( #StartUtility )
   END_RUNG
   RUNG wire#w1
      R_Coil( #StartChilling )
   END_RUNG
   RUNG wire#w1
      R_Coil( #StartBrine )
   END_RUNG
   RUNG wire#w1
      R_Coil( #StartJacketAirPurging )
   END_RUNG
   RUNG wire#w1
      R_Coil( #HeatTempReached )
   END_RUNG
   RUNG wire#w1
      R_Coil( #CoolTempReached )
   END_RUNG
   RUNG wire#w1
      { S7_GenerateENO := "TRUE" } Move(in := 0, out1 => #TimeMinPV)
   END_RUNG
   RUNG wire#w1
      { S7_GenerateENO := "TRUE" } Move(in := 0, out1 => #TimeSecPV)
   END_RUNG
   // the same network as SCL:
   IF (NOT #StartJacketAirPurging AND #Reset) OR NOT #Enable OR #Over THEN
       #Selected := FALSE;
       #Temp := FALSE;
       #JacketPressureReached := FALSE;
       #StartConfirmationPopupTemp := FALSE;
       #EndConfirmationPopupTemp := FALSE;
       #Started := FALSE;
       #StartJVDelay := FALSE;
       #StartJDDelay := FALSE;
       #StartUtility := FALSE;
       #StartChilling := FALSE;
       #StartBrine := FALSE;
   END_IF;
   #_w1 := (NOT #StartJacketAirPurging AND #Reset) OR NOT #Enable OR #Over;
   IF #_w1 THEN
       #StartJacketAirPurging := FALSE;
       #HeatTempReached := FALSE;
       #CoolTempReached := FALSE;
       #TimeMinPV := 0;
       #TimeSecPV := 0;
   END_IF;
END_REGION
END_FUNCTION_BLOCK

FUNCTION_BLOCK "FB103"   // FB103, LAD
TITLE = FB103
{ S7_Optimized_Access := 'FALSE' }
// ON DELAY TIMER (Retentive)
// stored: AutoNumber false, SetENOAutomatically false
   VAR_INPUT
      Enable : Bool;
      Running : Bool;
      SecPulse : Bool;
      AlwaysTrue : Bool;
      TimeSec : Int;
   END_VAR
   VAR_OUTPUT
      TimeOver : Bool;
      TimeSecPV : Int;
   END_VAR
   VAR_IN_OUT
      TimeOverTemp : Bool;
      TimeSecAct : Int;
   END_VAR
   VAR_TEMP   // added for the SCL form of the ladder/FBD networks
      _w1 : Bool;
   END_VAR
BEGIN

REGION Network 1: Timer On
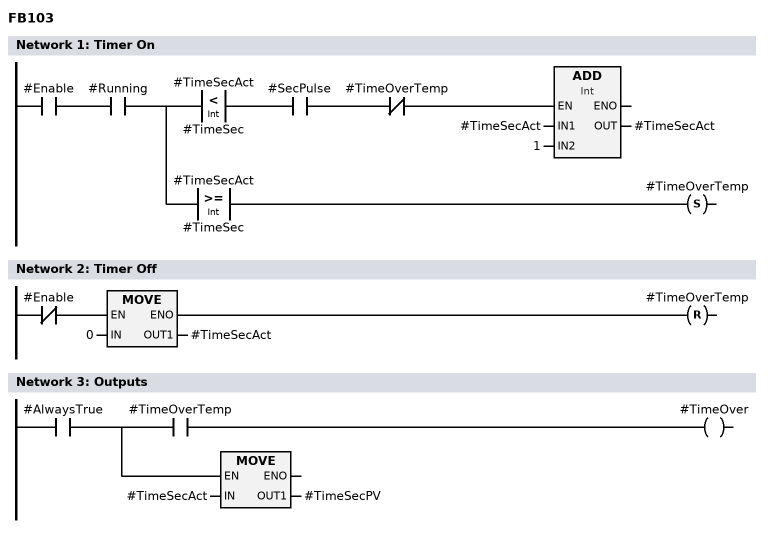
   RUNG wire#powerrail
      Contact( #Enable )
      Contact( #Running )
      wire#w1
      { S7_Templates := "SrcType := Int" } LT_Contact(in1 := #TimeSecAct, in2 := #TimeSec)
      Contact( #SecPulse )
      I_Contact( #TimeOverTemp )
      { S7_Templates := "SrcType := Int"; S7_GenerateENO := "TRUE" } Add(in1 := #TimeSecAct, in2 := 1, out => #TimeSecAct)
   END_RUNG
   RUNG wire#w1
      { S7_Templates := "SrcType := Int" } GE_Contact(in1 := #TimeSecAct, in2 := #TimeSec)
      S_Coil( #TimeOverTemp )
   END_RUNG
   // the same network as SCL:
   #_w1 := #Enable AND #Running;
   IF #_w1 AND (#TimeSecAct < #TimeSec) AND #SecPulse AND NOT #TimeOverTemp THEN
       #TimeSecAct := #TimeSecAct + 1;
   END_IF;
   IF #_w1 AND (#TimeSecAct >= #TimeSec) THEN #TimeOverTemp := TRUE; END_IF;
END_REGION

REGION Network 2: Timer Off
   RUNG wire#powerrail
      I_Contact( #Enable )
      { S7_GenerateENO := "TRUE" } Move(in := 0, out1 => #TimeSecAct)
      R_Coil( #TimeOverTemp )
   END_RUNG
   // the same network as SCL:
   // ENO of a box is taken as its EN; it also drops when the box reports an error
   IF NOT #Enable THEN
       #TimeSecAct := 0;
       #TimeOverTemp := FALSE;
   END_IF;
END_REGION

REGION Network 3: Outputs
   RUNG wire#powerrail
      Contact( #AlwaysTrue )
      wire#w1
      Contact( #TimeOverTemp )
      Coil( #TimeOver )
   END_RUNG
   RUNG wire#w1
      Move(in := #TimeSecAct, out1 => #TimeSecPV)
   END_RUNG
   // the same network as SCL:
   #TimeOver := #AlwaysTrue AND #TimeOverTemp;
   IF #AlwaysTrue THEN #TimeSecPV := #TimeSecAct; END_IF;
END_REGION
END_FUNCTION_BLOCK

FUNCTION_BLOCK "FB104"   // FB104, LAD
TITLE = FB104
{ S7_Optimized_Access := 'FALSE' }
// MANUAL PID
// stored: AutoNumber false, SetENOAutomatically false
   VAR_INPUT
      Enable : Bool;
      SecPulse : Bool;
      AlwaysTrue : Bool;
      DigitalOrAnalog : Bool;   // 0: DIGITAL; 1: ANALOG
      InvertPIDSel : Bool;   // 0: NO; 1: YES
      ActValue : Real;
      SetValue : Real;
      SetPoint1 : Real := 5.0;
      SetPoint2 : Real := 10.0;
      SetPoint3 : Real := 15.0;
      SetPoint4 : Real := 20.0;
      SetPoint5 : Real := 25.0;
      SetPoint6 : Real := 30.0;
      SetPoint7 : Real := 35.0;
      SetPoint8 : Real := 40.0;
      SetPoint9 : Real := 45.0;
      SetPoint10 : Real := 50.0;
      SetRef1 : Real := 10.0;
      SetRef2 : Real := 20.0;
      SetRef3 : Real := 30.0;
      SetRef4 : Real := 40.0;
      SetRef5 : Real := 50.0;
      SetRef6 : Real := 60.0;
      SetRef7 : Real := 70.0;
      SetRef8 : Real := 80.0;
      SetRef9 : Real := 90.0;
      SetRef10 : Real := 100.0;
      OnTime1 : Int := 2;
      OnTime2 : Int := 2;
      OnTime3 : Int := 2;
      OnTime4 : Int := 2;
      OnTime5 : Int := 2;
      OnTime6 : Int := 2;
      OnTime7 : Int := 2;
      OnTime8 : Int := 2;
      OnTime9 : Int := 2;
      OnTime10 : Int := 2;
      OffTime1 : Int := 3;
      OffTime2 : Int := 3;
      OffTime3 : Int := 3;
      OffTime4 : Int := 3;
      OffTime5 : Int := 3;
      OffTime6 : Int := 3;
      OffTime7 : Int := 3;
      OffTime8 : Int := 3;
      OffTime9 : Int := 3;
      OffTime10 : Int := 3;
   END_VAR
   VAR_OUTPUT
      Valve : Bool;
      SetRef : Real;
   END_VAR
   VAR_IN_OUT
      ControlValue1 : Real;
      ControlValue2 : Real;
      ControlValue3 : Real;
      ControlValue4 : Real;
      ControlValue5 : Real;
      ControlValue6 : Real;
      ControlValue7 : Real;
      ControlValue8 : Real;
      ControlValue9 : Real;
      ControlValue10 : Real;
   END_VAR
   VAR
      OnOffDelay { S7_SetPoint := 'True'} : "FB102";
      OnTime : Int;
      OffTime : Int;
   END_VAR
   VAR_TEMP   // added for the SCL form of the ladder/FBD networks
      _w1 : Bool;
   END_VAR
BEGIN

REGION Network 1: Set Point Calculations
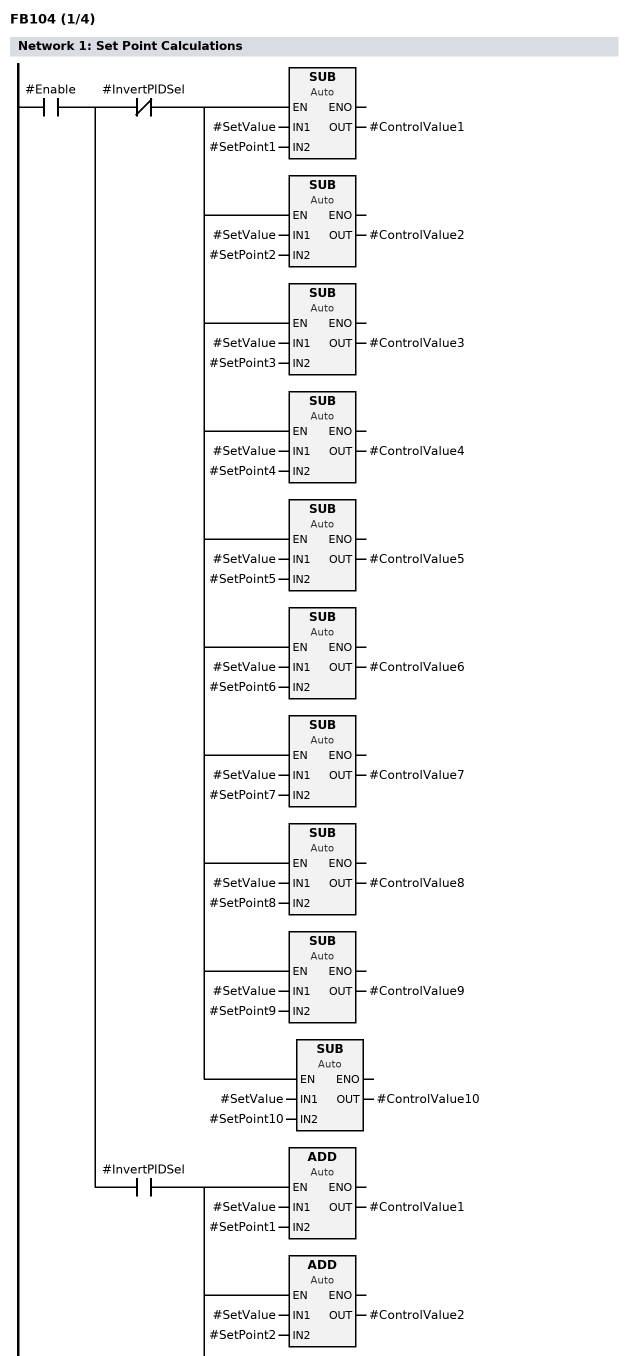
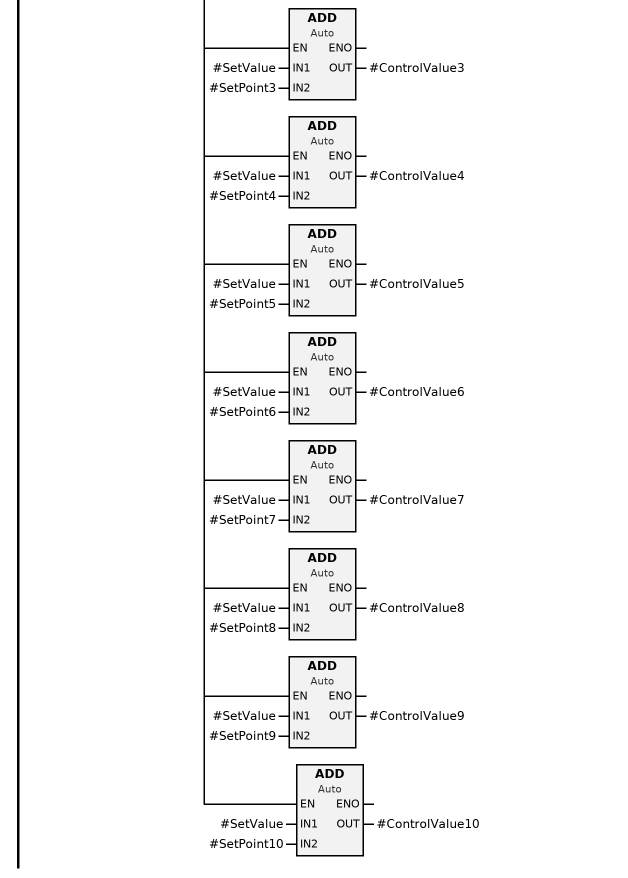
   RUNG wire#powerrail
      Contact( #Enable )
      wire#w1
      I_Contact( #InvertPIDSel )
      wire#w2
      Sub(in1 := #SetValue, in2 := #SetPoint1, out => #ControlValue1)
   END_RUNG
   RUNG wire#w2
      Sub(in1 := #SetValue, in2 := #SetPoint2, out => #ControlValue2)
   END_RUNG
   RUNG wire#w2
      Sub(in1 := #SetValue, in2 := #SetPoint3, out => #ControlValue3)
   END_RUNG
   RUNG wire#w2
      Sub(in1 := #SetValue, in2 := #SetPoint4, out => #ControlValue4)
   END_RUNG
   RUNG wire#w2
      Sub(in1 := #SetValue, in2 := #SetPoint5, out => #ControlValue5)
   END_RUNG
   RUNG wire#w2
      Sub(in1 := #SetValue, in2 := #SetPoint6, out => #ControlValue6)
   END_RUNG
   RUNG wire#w2
      Sub(in1 := #SetValue, in2 := #SetPoint7, out => #ControlValue7)
   END_RUNG
   RUNG wire#w2
      Sub(in1 := #SetValue, in2 := #SetPoint8, out => #ControlValue8)
   END_RUNG
   RUNG wire#w2
      Sub(in1 := #SetValue, in2 := #SetPoint9, out => #ControlValue9)
   END_RUNG
   RUNG wire#w2
      Sub(in1 := #SetValue, in2 := #SetPoint10, out => #ControlValue10)
   END_RUNG
   RUNG wire#w1
      Contact( #InvertPIDSel )
      wire#w3
      Add(in1 := #SetValue, in2 := #SetPoint1, out => #ControlValue1)
   END_RUNG
   RUNG wire#w3
      Add(in1 := #SetValue, in2 := #SetPoint2, out => #ControlValue2)
   END_RUNG
   RUNG wire#w3
      Add(in1 := #SetValue, in2 := #SetPoint3, out => #ControlValue3)
   END_RUNG
   RUNG wire#w3
      Add(in1 := #SetValue, in2 := #SetPoint4, out => #ControlValue4)
   END_RUNG
   RUNG wire#w3
      Add(in1 := #SetValue, in2 := #SetPoint5, out => #ControlValue5)
   END_RUNG
   RUNG wire#w3
      Add(in1 := #SetValue, in2 := #SetPoint6, out => #ControlValue6)
   END_RUNG
   RUNG wire#w3
      Add(in1 := #SetValue, in2 := #SetPoint7, out => #ControlValue7)
   END_RUNG
   RUNG wire#w3
      Add(in1 := #SetValue, in2 := #SetPoint8, out => #ControlValue8)
   END_RUNG
   RUNG wire#w3
      Add(in1 := #SetValue, in2 := #SetPoint9, out => #ControlValue9)
   END_RUNG
   RUNG wire#w3
      Add(in1 := #SetValue, in2 := #SetPoint10, out => #ControlValue10)
   END_RUNG
   // the same network as SCL:
   IF #Enable AND NOT #InvertPIDSel THEN
       #ControlValue1 := #SetValue - #SetPoint1;
       #ControlValue2 := #SetValue - #SetPoint2;
       #ControlValue3 := #SetValue - #SetPoint3;
       #ControlValue4 := #SetValue - #SetPoint4;
       #ControlValue5 := #SetValue - #SetPoint5;
       #ControlValue6 := #SetValue - #SetPoint6;
       #ControlValue7 := #SetValue - #SetPoint7;
       #ControlValue8 := #SetValue - #SetPoint8;
       #ControlValue9 := #SetValue - #SetPoint9;
       #ControlValue10 := #SetValue - #SetPoint10;
   END_IF;
   IF #Enable AND #InvertPIDSel THEN
       #ControlValue1 := #SetValue + #SetPoint1;
       #ControlValue2 := #SetValue + #SetPoint2;
       #ControlValue3 := #SetValue + #SetPoint3;
       #ControlValue4 := #SetValue + #SetPoint4;
       #ControlValue5 := #SetValue + #SetPoint5;
       #ControlValue6 := #SetValue + #SetPoint6;
       #ControlValue7 := #SetValue + #SetPoint7;
       #ControlValue8 := #SetValue + #SetPoint8;
       #ControlValue9 := #SetValue + #SetPoint9;
       #ControlValue10 := #SetValue + #SetPoint10;
   END_IF;
END_REGION

REGION Network 2: Set Reference for InvertPIDSel: NO
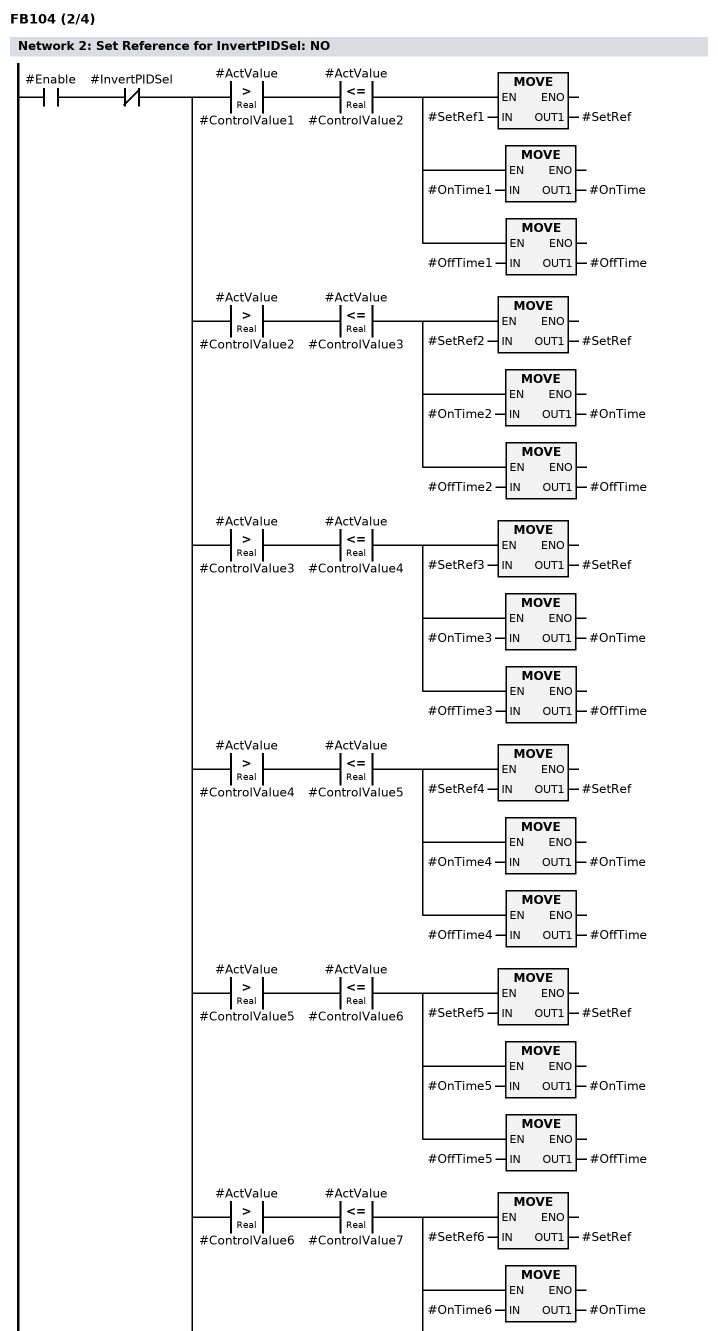
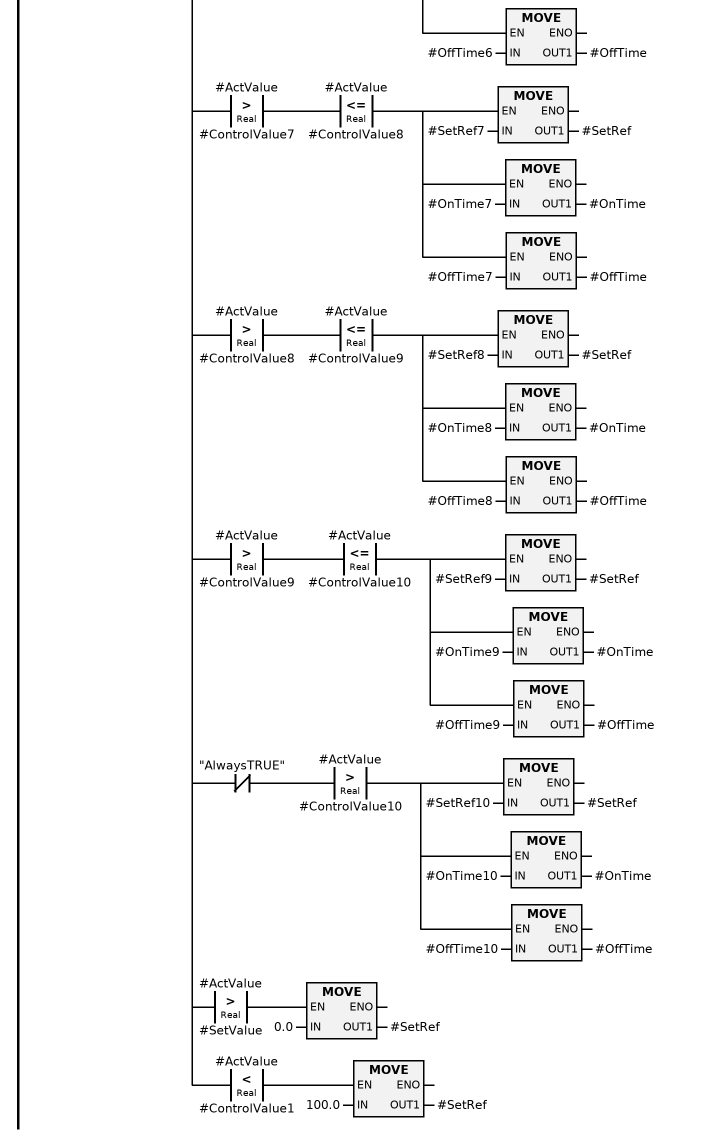
   RUNG wire#powerrail
      Contact( #Enable )
      I_Contact( #InvertPIDSel )
      wire#w1
      { S7_Templates := "SrcType := Real" } GT_Contact(in1 := #ActValue, in2 := #ControlValue1)
      { S7_Templates := "SrcType := Real" } LE_Contact(in1 := #ActValue, in2 := #ControlValue2)
      wire#w2
      Move(in := #SetRef1, out1 => #SetRef)
   END_RUNG
   RUNG wire#w2
      Move(in := #OnTime1, out1 => #OnTime)
   END_RUNG
   RUNG wire#w2
      Move(in := #OffTime1, out1 => #OffTime)
   END_RUNG
   RUNG wire#w1
      { S7_Templates := "SrcType := Real" } GT_Contact(in1 := #ActValue, in2 := #ControlValue2)
      { S7_Templates := "SrcType := Real" } LE_Contact(in1 := #ActValue, in2 := #ControlValue3)
      wire#w3
      Move(in := #SetRef2, out1 => #SetRef)
   END_RUNG
   RUNG wire#w3
      Move(in := #OnTime2, out1 => #OnTime)
   END_RUNG
   RUNG wire#w3
      Move(in := #OffTime2, out1 => #OffTime)
   END_RUNG
   RUNG wire#w1
      { S7_Templates := "SrcType := Real" } GT_Contact(in1 := #ActValue, in2 := #ControlValue3)
      { S7_Templates := "SrcType := Real" } LE_Contact(in1 := #ActValue, in2 := #ControlValue4)
      wire#w4
      Move(in := #SetRef3, out1 => #SetRef)
   END_RUNG
   RUNG wire#w4
      Move(in := #OnTime3, out1 => #OnTime)
   END_RUNG
   RUNG wire#w4
      Move(in := #OffTime3, out1 => #OffTime)
   END_RUNG
   RUNG wire#w1
      { S7_Templates := "SrcType := Real" } GT_Contact(in1 := #ActValue, in2 := #ControlValue4)
      { S7_Templates := "SrcType := Real" } LE_Contact(in1 := #ActValue, in2 := #ControlValue5)
      wire#w5
      Move(in := #SetRef4, out1 => #SetRef)
   END_RUNG
   RUNG wire#w5
      Move(in := #OnTime4, out1 => #OnTime)
   END_RUNG
   RUNG wire#w5
      Move(in := #OffTime4, out1 => #OffTime)
   END_RUNG
   RUNG wire#w1
      { S7_Templates := "SrcType := Real" } GT_Contact(in1 := #ActValue, in2 := #ControlValue5)
      { S7_Templates := "SrcType := Real" } LE_Contact(in1 := #ActValue, in2 := #ControlValue6)
      wire#w6
      Move(in := #SetRef5, out1 => #SetRef)
   END_RUNG
   RUNG wire#w6
      Move(in := #OnTime5, out1 => #OnTime)
   END_RUNG
   RUNG wire#w6
      Move(in := #OffTime5, out1 => #OffTime)
   END_RUNG
   RUNG wire#w1
      { S7_Templates := "SrcType := Real" } GT_Contact(in1 := #ActValue, in2 := #ControlValue6)
      { S7_Templates := "SrcType := Real" } LE_Contact(in1 := #ActValue, in2 := #ControlValue7)
      wire#w7
      Move(in := #SetRef6, out1 => #SetRef)
   END_RUNG
   RUNG wire#w7
      Move(in := #OnTime6, out1 => #OnTime)
   END_RUNG
   RUNG wire#w7
      Move(in := #OffTime6, out1 => #OffTime)
   END_RUNG
   RUNG wire#w1
      { S7_Templates := "SrcType := Real" } GT_Contact(in1 := #ActValue, in2 := #ControlValue7)
      { S7_Templates := "SrcType := Real" } LE_Contact(in1 := #ActValue, in2 := #ControlValue8)
      wire#w8
      Move(in := #SetRef7, out1 => #SetRef)
   END_RUNG
   RUNG wire#w8
      Move(in := #OnTime7, out1 => #OnTime)
   END_RUNG
   RUNG wire#w8
      Move(in := #OffTime7, out1 => #OffTime)
   END_RUNG
   RUNG wire#w1
      { S7_Templates := "SrcType := Real" } GT_Contact(in1 := #ActValue, in2 := #ControlValue8)
      { S7_Templates := "SrcType := Real" } LE_Contact(in1 := #ActValue, in2 := #ControlValue9)
      wire#w9
      Move(in := #SetRef8, out1 => #SetRef)
   END_RUNG
   RUNG wire#w9
      Move(in := #OnTime8, out1 => #OnTime)
   END_RUNG
   RUNG wire#w9
      Move(in := #OffTime8, out1 => #OffTime)
   END_RUNG
   RUNG wire#w1
      { S7_Templates := "SrcType := Real" } GT_Contact(in1 := #ActValue, in2 := #ControlValue9)
      { S7_Templates := "SrcType := Real" } LE_Contact(in1 := #ActValue, in2 := #ControlValue10)
      wire#w10
      Move(in := #SetRef9, out1 => #SetRef)
   END_RUNG
   RUNG wire#w10
      Move(in := #OnTime9, out1 => #OnTime)
   END_RUNG
   RUNG wire#w10
      Move(in := #OffTime9, out1 => #OffTime)
   END_RUNG
   RUNG wire#w1
      I_Contact( "AlwaysTRUE" )
      { S7_Templates := "SrcType := Real" } GT_Contact(in1 := #ActValue, in2 := #ControlValue10)
      wire#w11
      Move(in := #SetRef10, out1 => #SetRef)
   END_RUNG
   RUNG wire#w11
      Move(in := #OnTime10, out1 => #OnTime)
   END_RUNG
   RUNG wire#w11
      Move(in := #OffTime10, out1 => #OffTime)
   END_RUNG
   RUNG wire#w1
      { S7_Templates := "SrcType := Real" } GT_Contact(in1 := #ActValue, in2 := #SetValue)
      Move(in := 0.0, out1 => #SetRef)
   END_RUNG
   RUNG wire#w1
      { S7_Templates := "SrcType := Real" } LT_Contact(in1 := #ActValue, in2 := #ControlValue1)
      Move(in := 100.0, out1 => #SetRef)
   END_RUNG
   // the same network as SCL:
   #_w1 := #Enable AND NOT #InvertPIDSel;
   IF #_w1 AND (#ActValue > #ControlValue1) AND (#ActValue <= #ControlValue2) THEN
       #SetRef := #SetRef1;
       #OnTime := #OnTime1;
       #OffTime := #OffTime1;
   END_IF;
   IF #_w1 AND (#ActValue > #ControlValue2) AND (#ActValue <= #ControlValue3) THEN
       #SetRef := #SetRef2;
       #OnTime := #OnTime2;
       #OffTime := #OffTime2;
   END_IF;
   IF #_w1 AND (#ActValue > #ControlValue3) AND (#ActValue <= #ControlValue4) THEN
       #SetRef := #SetRef3;
       #OnTime := #OnTime3;
       #OffTime := #OffTime3;
   END_IF;
   IF #_w1 AND (#ActValue > #ControlValue4) AND (#ActValue <= #ControlValue5) THEN
       #SetRef := #SetRef4;
       #OnTime := #OnTime4;
       #OffTime := #OffTime4;
   END_IF;
   IF #_w1 AND (#ActValue > #ControlValue5) AND (#ActValue <= #ControlValue6) THEN
       #SetRef := #SetRef5;
       #OnTime := #OnTime5;
       #OffTime := #OffTime5;
   END_IF;
   IF #_w1 AND (#ActValue > #ControlValue6) AND (#ActValue <= #ControlValue7) THEN
       #SetRef := #SetRef6;
       #OnTime := #OnTime6;
       #OffTime := #OffTime6;
   END_IF;
   IF #_w1 AND (#ActValue > #ControlValue7) AND (#ActValue <= #ControlValue8) THEN
       #SetRef := #SetRef7;
       #OnTime := #OnTime7;
       #OffTime := #OffTime7;
   END_IF;
   IF #_w1 AND (#ActValue > #ControlValue8) AND (#ActValue <= #ControlValue9) THEN
       #SetRef := #SetRef8;
       #OnTime := #OnTime8;
       #OffTime := #OffTime8;
   END_IF;
   IF #_w1 AND (#ActValue > #ControlValue9) AND (#ActValue <= #ControlValue10) THEN
       #SetRef := #SetRef9;
       #OnTime := #OnTime9;
       #OffTime := #OffTime9;
   END_IF;
   IF #_w1 AND NOT "AlwaysTRUE" AND (#ActValue > #ControlValue10) THEN
       #SetRef := #SetRef10;
       #OnTime := #OnTime10;
       #OffTime := #OffTime10;
   END_IF;
   IF #_w1 AND (#ActValue > #SetValue) THEN #SetRef := 0.0; END_IF;
   IF #_w1 AND (#ActValue < #ControlValue1) THEN #SetRef := 100.0; END_IF;
END_REGION

REGION Network 3: Set Reference for InvertPIDSel: YES
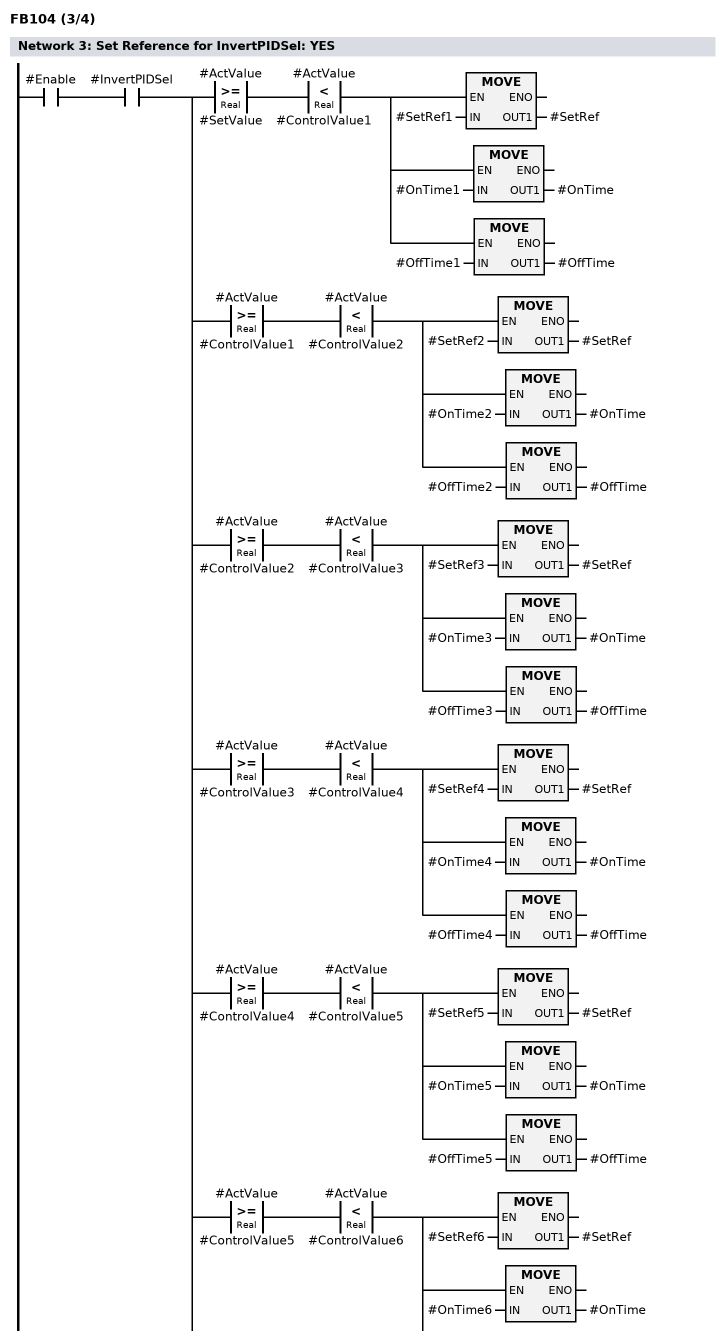
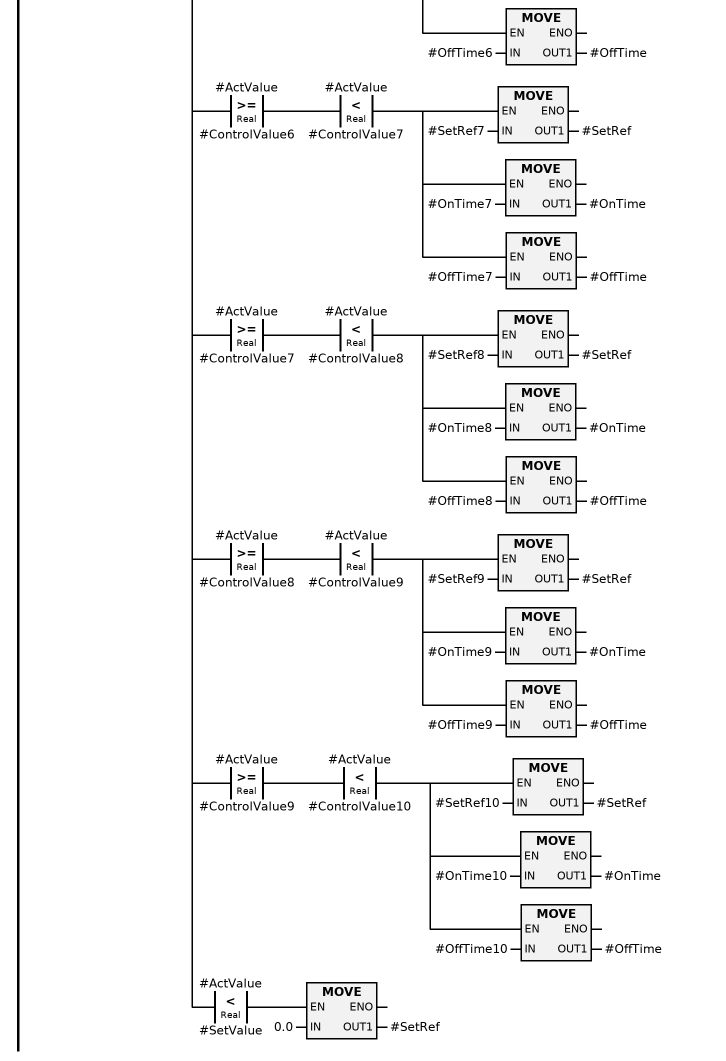
   RUNG wire#powerrail
      Contact( #Enable )
      Contact( #InvertPIDSel )
      wire#w1
      { S7_Templates := "SrcType := Real" } GE_Contact(in1 := #ActValue, in2 := #SetValue)
      { S7_Templates := "SrcType := Real" } LT_Contact(in1 := #ActValue, in2 := #ControlValue1)
      wire#w2
      Move(in := #SetRef1, out1 => #SetRef)
   END_RUNG
   RUNG wire#w2
      Move(in := #OnTime1, out1 => #OnTime)
   END_RUNG
   RUNG wire#w2
      Move(in := #OffTime1, out1 => #OffTime)
   END_RUNG
   RUNG wire#w1
      { S7_Templates := "SrcType := Real" } GE_Contact(in1 := #ActValue, in2 := #ControlValue1)
      { S7_Templates := "SrcType := Real" } LT_Contact(in1 := #ActValue, in2 := #ControlValue2)
      wire#w3
      Move(in := #SetRef2, out1 => #SetRef)
   END_RUNG
   RUNG wire#w3
      Move(in := #OnTime2, out1 => #OnTime)
   END_RUNG
   RUNG wire#w3
      Move(in := #OffTime2, out1 => #OffTime)
   END_RUNG
   RUNG wire#w1
      { S7_Templates := "SrcType := Real" } GE_Contact(in1 := #ActValue, in2 := #ControlValue2)
      { S7_Templates := "SrcType := Real" } LT_Contact(in1 := #ActValue, in2 := #ControlValue3)
      wire#w4
      Move(in := #SetRef3, out1 => #SetRef)
   END_RUNG
   RUNG wire#w4
      Move(in := #OnTime3, out1 => #OnTime)
   END_RUNG
   RUNG wire#w4
      Move(in := #OffTime3, out1 => #OffTime)
   END_RUNG
   RUNG wire#w1
      { S7_Templates := "SrcType := Real" } GE_Contact(in1 := #ActValue, in2 := #ControlValue3)
      { S7_Templates := "SrcType := Real" } LT_Contact(in1 := #ActValue, in2 := #ControlValue4)
      wire#w5
      Move(in := #SetRef4, out1 => #SetRef)
   END_RUNG
   RUNG wire#w5
      Move(in := #OnTime4, out1 => #OnTime)
   END_RUNG
   RUNG wire#w5
      Move(in := #OffTime4, out1 => #OffTime)
   END_RUNG
   RUNG wire#w1
      { S7_Templates := "SrcType := Real" } GE_Contact(in1 := #ActValue, in2 := #ControlValue4)
      { S7_Templates := "SrcType := Real" } LT_Contact(in1 := #ActValue, in2 := #ControlValue5)
      wire#w6
      Move(in := #SetRef5, out1 => #SetRef)
   END_RUNG
   RUNG wire#w6
      Move(in := #OnTime5, out1 => #OnTime)
   END_RUNG
   RUNG wire#w6
      Move(in := #OffTime5, out1 => #OffTime)
   END_RUNG
   RUNG wire#w1
      { S7_Templates := "SrcType := Real" } GE_Contact(in1 := #ActValue, in2 := #ControlValue5)
      { S7_Templates := "SrcType := Real" } LT_Contact(in1 := #ActValue, in2 := #ControlValue6)
      wire#w7
      Move(in := #SetRef6, out1 => #SetRef)
   END_RUNG
   RUNG wire#w7
      Move(in := #OnTime6, out1 => #OnTime)
   END_RUNG
   RUNG wire#w7
      Move(in := #OffTime6, out1 => #OffTime)
   END_RUNG
   RUNG wire#w1
      { S7_Templates := "SrcType := Real" } GE_Contact(in1 := #ActValue, in2 := #ControlValue6)
      { S7_Templates := "SrcType := Real" } LT_Contact(in1 := #ActValue, in2 := #ControlValue7)
      wire#w8
      Move(in := #SetRef7, out1 => #SetRef)
   END_RUNG
   RUNG wire#w8
      Move(in := #OnTime7, out1 => #OnTime)
   END_RUNG
   RUNG wire#w8
      Move(in := #OffTime7, out1 => #OffTime)
   END_RUNG
   RUNG wire#w1
      { S7_Templates := "SrcType := Real" } GE_Contact(in1 := #ActValue, in2 := #ControlValue7)
      { S7_Templates := "SrcType := Real" } LT_Contact(in1 := #ActValue, in2 := #ControlValue8)
      wire#w9
      Move(in := #SetRef8, out1 => #SetRef)
   END_RUNG
   RUNG wire#w9
      Move(in := #OnTime8, out1 => #OnTime)
   END_RUNG
   RUNG wire#w9
      Move(in := #OffTime8, out1 => #OffTime)
   END_RUNG
   RUNG wire#w1
      { S7_Templates := "SrcType := Real" } GE_Contact(in1 := #ActValue, in2 := #ControlValue8)
      { S7_Templates := "SrcType := Real" } LT_Contact(in1 := #ActValue, in2 := #ControlValue9)
      wire#w10
      Move(in := #SetRef9, out1 => #SetRef)
   END_RUNG
   RUNG wire#w10
      Move(in := #OnTime9, out1 => #OnTime)
   END_RUNG
   RUNG wire#w10
      Move(in := #OffTime9, out1 => #OffTime)
   END_RUNG
   RUNG wire#w1
      { S7_Templates := "SrcType := Real" } GE_Contact(in1 := #ActValue, in2 := #ControlValue9)
      { S7_Templates := "SrcType := Real" } LT_Contact(in1 := #ActValue, in2 := #ControlValue10)
      wire#w11
      Move(in := #SetRef10, out1 => #SetRef)
   END_RUNG
   RUNG wire#w11
      Move(in := #OnTime10, out1 => #OnTime)
   END_RUNG
   RUNG wire#w11
      Move(in := #OffTime10, out1 => #OffTime)
   END_RUNG
   RUNG wire#w1
      { S7_Templates := "SrcType := Real" } LT_Contact(in1 := #ActValue, in2 := #SetValue)
      Move(in := 0.0, out1 => #SetRef)
   END_RUNG
   // the same network as SCL:
   #_w1 := #Enable AND #InvertPIDSel;
   IF #_w1 AND (#ActValue >= #SetValue) AND (#ActValue < #ControlValue1) THEN
       #SetRef := #SetRef1;
       #OnTime := #OnTime1;
       #OffTime := #OffTime1;
   END_IF;
   IF #_w1 AND (#ActValue >= #ControlValue1) AND (#ActValue < #ControlValue2) THEN
       #SetRef := #SetRef2;
       #OnTime := #OnTime2;
       #OffTime := #OffTime2;
   END_IF;
   IF #_w1 AND (#ActValue >= #ControlValue2) AND (#ActValue < #ControlValue3) THEN
       #SetRef := #SetRef3;
       #OnTime := #OnTime3;
       #OffTime := #OffTime3;
   END_IF;
   IF #_w1 AND (#ActValue >= #ControlValue3) AND (#ActValue < #ControlValue4) THEN
       #SetRef := #SetRef4;
       #OnTime := #OnTime4;
       #OffTime := #OffTime4;
   END_IF;
   IF #_w1 AND (#ActValue >= #ControlValue4) AND (#ActValue < #ControlValue5) THEN
       #SetRef := #SetRef5;
       #OnTime := #OnTime5;
       #OffTime := #OffTime5;
   END_IF;
   IF #_w1 AND (#ActValue >= #ControlValue5) AND (#ActValue < #ControlValue6) THEN
       #SetRef := #SetRef6;
       #OnTime := #OnTime6;
       #OffTime := #OffTime6;
   END_IF;
   IF #_w1 AND (#ActValue >= #ControlValue6) AND (#ActValue < #ControlValue7) THEN
       #SetRef := #SetRef7;
       #OnTime := #OnTime7;
       #OffTime := #OffTime7;
   END_IF;
   IF #_w1 AND (#ActValue >= #ControlValue7) AND (#ActValue < #ControlValue8) THEN
       #SetRef := #SetRef8;
       #OnTime := #OnTime8;
       #OffTime := #OffTime8;
   END_IF;
   IF #_w1 AND (#ActValue >= #ControlValue8) AND (#ActValue < #ControlValue9) THEN
       #SetRef := #SetRef9;
       #OnTime := #OnTime9;
       #OffTime := #OffTime9;
   END_IF;
   IF #_w1 AND (#ActValue >= #ControlValue9) AND (#ActValue < #ControlValue10) THEN
       #SetRef := #SetRef10;
       #OnTime := #OnTime10;
       #OffTime := #OffTime10;
   END_IF;
   IF #_w1 AND (#ActValue < #SetValue) THEN #SetRef := 0.0; END_IF;
END_REGION

REGION Network 4: On/Off Delay
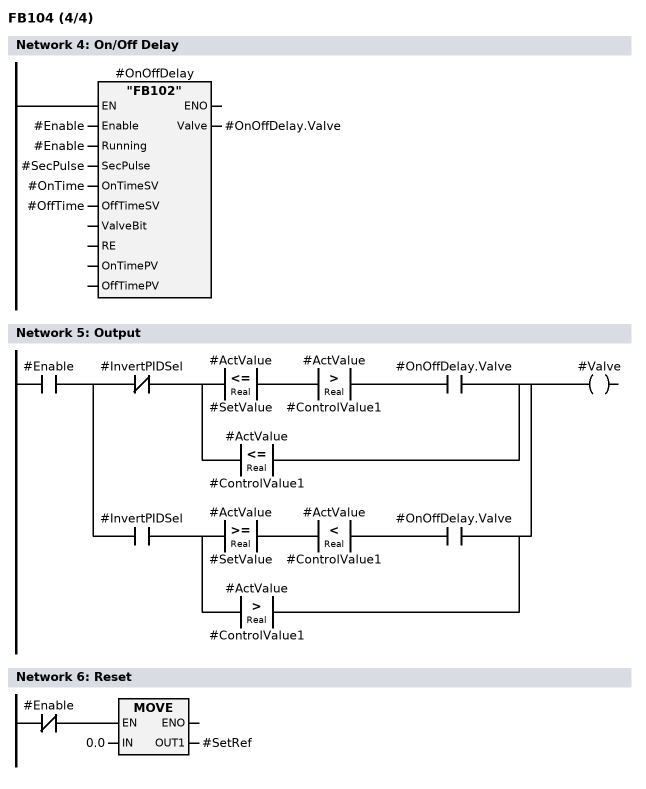
   RUNG wire#powerrail
      #OnOffDelay(Enable := #Enable, Running := #Enable, SecPulse := #SecPulse, OnTimeSV := #OnTime, OffTimeSV := #OffTime, ValveBit :=, RE :=, OnTimePV :=, OffTimePV :=, Valve => #OnOffDelay.Valve)
   END_RUNG
   // the same network as SCL:
   #OnOffDelay(Enable := #Enable,   // "FB102"
               Running := #Enable,
               SecPulse := #SecPulse,
               OnTimeSV := #OnTime,
               OffTimeSV := #OffTime,
               Valve => #OnOffDelay.Valve);
END_REGION

REGION Network 5: Output
   RUNG wire#powerrail
      Contact( #Enable )
      wire#w1
      I_Contact( #InvertPIDSel )
      wire#w2
      { S7_Templates := "SrcType := Real" } LE_Contact(in1 := #ActValue, in2 := #SetValue)
      { S7_Templates := "SrcType := Real" } GT_Contact(in1 := #ActValue, in2 := #ControlValue1)
      Contact( #OnOffDelay.Valve )
      wire#w3
      Coil( #Valve )
   END_RUNG
   RUNG wire#w2
      { S7_Templates := "SrcType := Real" } LE_Contact(in1 := #ActValue, in2 := #ControlValue1)
   END_RUNG wire#w3
   RUNG wire#w1
      Contact( #InvertPIDSel )
      wire#w4
      { S7_Templates := "SrcType := Real" } GE_Contact(in1 := #ActValue, in2 := #SetValue)
      { S7_Templates := "SrcType := Real" } LT_Contact(in1 := #ActValue, in2 := #ControlValue1)
      Contact( #OnOffDelay.Valve )
   END_RUNG wire#w3
   RUNG wire#w4
      { S7_Templates := "SrcType := Real" } GT_Contact(in1 := #ActValue, in2 := #ControlValue1)
   END_RUNG wire#w3
   // the same network as SCL:
   #Valve := #Enable AND ((NOT #InvertPIDSel AND (((#ActValue <= #SetValue) AND (#ActValue > #ControlValue1) AND #OnOffDelay.Valve) OR (#ActValue <= #ControlValue1))) OR (#InvertPIDSel AND (((#ActValue >= #SetValue) AND (#ActValue < #ControlValue1) AND #OnOffDelay.Valve) OR (#ActValue > #ControlValue1))));
END_REGION

REGION Network 6: Reset
   RUNG wire#powerrail
      I_Contact( #Enable )
      Move(in := 0.0, out1 => #SetRef)
   END_RUNG
   // the same network as SCL:
   IF NOT #Enable THEN #SetRef := 0.0; END_IF;
END_REGION
END_FUNCTION_BLOCK

FUNCTION_BLOCK "FB302"   // FB302, LAD
TITLE = FB302
{ S7_Optimized_Access := 'TRUE' }
AUTHOR : PRECISE
FAMILY : PRECISE
// MIXING
// stored: AutoNumber false, MemoryReserve 100, SetENOAutomatically false
   VAR_INPUT
      Enable : Bool;
      Disable : Bool;
      Fault : Bool;
      SecPulse : Bool;
      AlwaysTrue : Bool;
      StartConfirmationPopupSel : Bool;   // StartConfirmationPopupSel: 0-NO/1-YES
      EndConfirmationPopupSel : Bool;   // EndConfirmationPopupSel: 0-NO/1-YES
      MixingModeSel : Int;   // Mixing Mode Selection: 0-Auto/1-Manual
      MixerTypeSel : Int;   // Mixer Type Selection: 0-MM/1-USM/2-HSM/3-BP/4-ANCHOR
      MixingTimeBaseSel : Bool;   // Mixing Time Base Selection: 0-second/1-minute
      MixingTimeMin : Int := 1;   // For Mixing Mode Selection: 0-Auto & Mixing Time Base Selection: 1-minute
      MixingTimeSec : Int := 30;   // For Mixing Mode Selection: 0-Auto & Mixing Time Base Selection: 0-second
      MixingSpeed : Real := 100.0;
   END_VAR
   VAR_OUTPUT
      MixerCmd : Bool;
      WaterInletValve : Bool;
      StartConfirmationPopup : Bool;   // For Start Confirmation Popup Selection: Yes
      EndConfirmationPopup : Bool;   // For End Confirmation Popup Selection: Yes
      ManualPopup : Bool;   // For Mixing Mode Selection: 1-Manual
      MixingTimeMinPV : DInt;   // For Mixing Mode Selection: 0-Auto
      MixingTimeSecPV : DInt;   // For Mixing Mode Selection: 0-Auto
      MixingSpeedPV : Real;
      PrintTrigger : Bool;
      PrintWord : Int;
      PrintStatus : String[50];
   END_VAR
   VAR_IN_OUT
      Start : Bool;
      Stop : Bool;
      Reset : Bool;
      StartConfirmationAck : Bool;   // For Start Confirmation Popup Selection: Yes
      EndConfirmationAck : Bool;   // For End Confirmation Popup Selection: Yes
      ManualAck : Bool;   // For Mixing Mode Selection: 1-Manual
      Cp01Fsc : Bool;
      SpareBtn2 : Bool;
      Running : Bool;
      Selected : Bool;
      Paused : Bool;
      StartConfirmationPopupTemp : Bool;   // For Start Confirmation Popup Selection: Yes
      EndConfirmationPopupTemp : Bool;   // For End Confirmation Popup Selection: Yes
      ManualPopupTemp : Bool;   // For Mixing Mode Selection: 1-Manual
      MixingStarted : Bool;
      MixingOver : Bool;
   END_VAR
   VAR
      PrintTriggerTemp : Bool;
      RE1 : Bool;
      RE2 : Bool;
      RE3 : Bool;
      RE4 : Bool;
      RE5 : Bool;
      RE6 : Bool;
      RE7 : Bool;
      MixingTimer : "FB101";
      PrintTriggerResetTimer { S7_SetPoint := 'True'} : TON_TIME;
      BtnResetTimer { S7_SetPoint := 'True'} : TON_TIME;
   END_VAR
   VAR_TEMP
      STATUS1 : String[40];
      STATUS2 : String[40];
      STATUS3 : String[40];
      STATUS4 : String[40];
      STATUS5 : String[40];
   END_VAR
   VAR_TEMP   // added for the SCL form of the ladder/FBD networks
      _w1 : Bool;
      _w2 : Bool;
      _w3 : Bool;
      _w4 : Bool;
      _w5 : Bool;
   END_VAR
BEGIN

REGION Network 1: Running
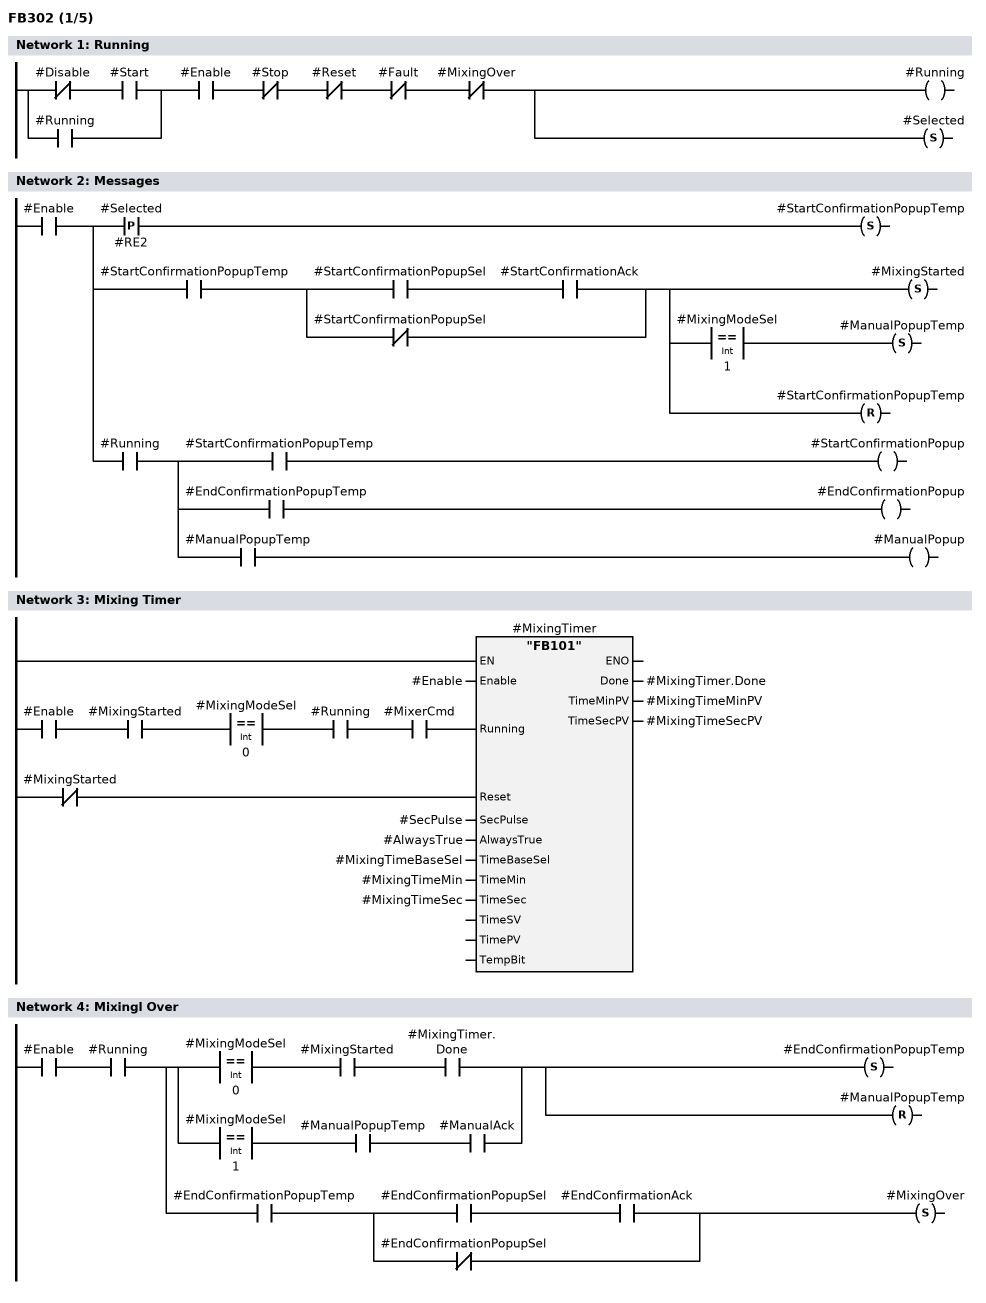
   RUNG wire#powerrail
      I_Contact( #Disable )
      Contact( #Start )
      wire#w1
      Contact( #Enable )
      I_Contact( #Stop )
      I_Contact( #Reset )
      I_Contact( #Fault )
      I_Contact( #MixingOver )
      wire#w2
      Coil( #Running )
   END_RUNG
   RUNG wire#powerrail
      Contact( #Running )
   END_RUNG wire#w1
   RUNG wire#w2
      S_Coil( #Selected )
   END_RUNG
   // the same network as SCL:
   #Running := ((NOT #Disable AND #Start) OR #Running) AND #Enable AND NOT #Stop AND NOT #Reset AND NOT #Fault AND NOT #MixingOver;
   IF #Running THEN #Selected := TRUE; END_IF;
END_REGION

REGION Network 2: Messages
   RUNG wire#powerrail
      Contact( #Enable )
      wire#w1
      P_Contact(operand := #Selected, bit := #RE2)
      S_Coil( #StartConfirmationPopupTemp )
   END_RUNG
   RUNG wire#w1
      Contact( #StartConfirmationPopupTemp )
      wire#w2
      Contact( #StartConfirmationPopupSel )
      Contact( #StartConfirmationAck )
      wire#w3
      S_Coil( #MixingStarted )
   END_RUNG
   RUNG wire#w2
      I_Contact( #StartConfirmationPopupSel )
   END_RUNG wire#w3
   RUNG wire#w3
      { S7_Templates := "SrcType := Int" } EQ_Contact(in1 := #MixingModeSel, in2 := 1)
      S_Coil( #ManualPopupTemp )
   END_RUNG
   RUNG wire#w3
      R_Coil( #StartConfirmationPopupTemp )
   END_RUNG
   RUNG wire#w1
      Contact( #Running )
      wire#w4
      Contact( #StartConfirmationPopupTemp )
      Coil( #StartConfirmationPopup )
   END_RUNG
   RUNG wire#w4
      Contact( #EndConfirmationPopupTemp )
      Coil( #EndConfirmationPopup )
   END_RUNG
   RUNG wire#w4
      Contact( #ManualPopupTemp )
      Coil( #ManualPopup )
   END_RUNG
   // the same network as SCL:
   #_w1 := #Enable AND #Selected AND NOT #RE2;   // rising edge of #Selected
   #RE2 := #Selected;
   IF #_w1 THEN #StartConfirmationPopupTemp := TRUE; END_IF;
   #_w2 := #Enable AND #StartConfirmationPopupTemp AND ((#StartConfirmationPopupSel AND #StartConfirmationAck) OR NOT #StartConfirmationPopupSel);
   IF #_w2 THEN #MixingStarted := TRUE; END_IF;
   IF #_w2 AND (#MixingModeSel = 1) THEN #ManualPopupTemp := TRUE; END_IF;
   IF #_w2 THEN #StartConfirmationPopupTemp := FALSE; END_IF;
   #_w3 := #Enable AND #Running;
   #StartConfirmationPopup := #_w3 AND #StartConfirmationPopupTemp;
   #EndConfirmationPopup := #_w3 AND #EndConfirmationPopupTemp;
   #ManualPopup := #_w3 AND #ManualPopupTemp;
END_REGION

REGION Network 3: Mixing Timer
   RUNG wire#powerrail
      #MixingTimer(Running := wire#w1, Reset := wire#w2, Enable := #Enable, SecPulse := #SecPulse, AlwaysTrue := #AlwaysTrue, TimeBaseSel := #MixingTimeBaseSel, TimeMin := #MixingTimeMin, TimeSec := #MixingTimeSec, TimeSV :=, TimePV :=, TempBit :=, Done => #MixingTimer.Done, TimeMinPV => #MixingTimeMinPV, TimeSecPV => #MixingTimeSecPV)
   END_RUNG
   RUNG wire#powerrail
      Contact( #Enable )
      Contact( #MixingStarted )
      { S7_Templates := "SrcType := Int" } EQ_Contact(in1 := #MixingModeSel, in2 := 0)
      Contact( #Running )
      Contact( #MixerCmd )
   END_RUNG wire#w1
   RUNG wire#powerrail
      I_Contact( #MixingStarted )
   END_RUNG wire#w2
   // the same network as SCL:
   #MixingTimer(Enable := #Enable,   // "FB101"
                Running := #Enable AND #MixingStarted AND (#MixingModeSel = 0) AND #Running AND #MixerCmd,
                Reset := NOT #MixingStarted,
                SecPulse := #SecPulse,
                AlwaysTrue := #AlwaysTrue,
                TimeBaseSel := #MixingTimeBaseSel,
                TimeMin := #MixingTimeMin,
                TimeSec := #MixingTimeSec,
                Done => #MixingTimer.Done,
                TimeMinPV => #MixingTimeMinPV,
                TimeSecPV => #MixingTimeSecPV);
END_REGION

REGION Network 4: Mixingl Over
   RUNG wire#powerrail
      Contact( #Enable )
      Contact( #Running )
      wire#w1
      { S7_Templates := "SrcType := Int" } EQ_Contact(in1 := #MixingModeSel, in2 := 0)
      Contact( #MixingStarted )
      Contact( #MixingTimer.Done )
      wire#w2
      S_Coil( #EndConfirmationPopupTemp )
   END_RUNG
   RUNG wire#w1
      { S7_Templates := "SrcType := Int" } EQ_Contact(in1 := #MixingModeSel, in2 := 1)
      Contact( #ManualPopupTemp )
      Contact( #ManualAck )
   END_RUNG wire#w2
   RUNG wire#w2
      R_Coil( #ManualPopupTemp )
   END_RUNG
   RUNG wire#w1
      Contact( #EndConfirmationPopupTemp )
      wire#w3
      Contact( #EndConfirmationPopupSel )
      Contact( #EndConfirmationAck )
      wire#w4
      S_Coil( #MixingOver )
   END_RUNG
   RUNG wire#w3
      I_Contact( #EndConfirmationPopupSel )
   END_RUNG wire#w4
   // the same network as SCL:
   #_w1 := #Enable AND #Running;
   IF #_w1 AND (((#MixingModeSel = 0) AND #MixingStarted AND #MixingTimer.Done) OR ((#MixingModeSel = 1) AND #ManualPopupTemp AND #ManualAck)) THEN
       #EndConfirmationPopupTemp := TRUE;
       #ManualPopupTemp := FALSE;
   END_IF;
   IF #_w1 AND #EndConfirmationPopupTemp AND ((#EndConfirmationPopupSel AND #EndConfirmationAck) OR NOT #EndConfirmationPopupSel) THEN
       #MixingOver := TRUE;
   END_IF;
END_REGION

REGION Network 5: Output On
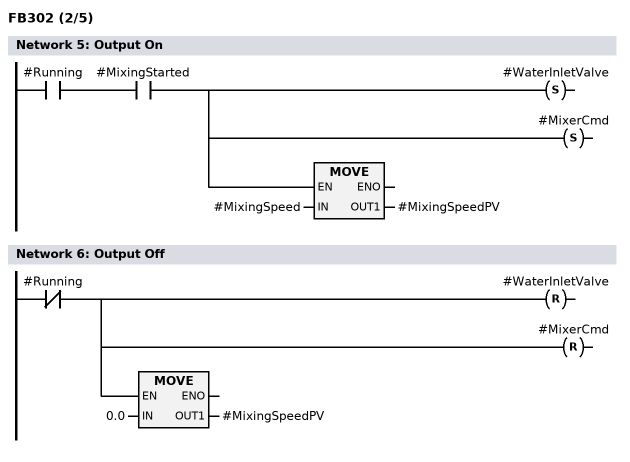
   RUNG wire#powerrail
      Contact( #Running )
      Contact( #MixingStarted )
      wire#w1
      S_Coil( #WaterInletValve )
   END_RUNG
   RUNG wire#w1
      S_Coil( #MixerCmd )
   END_RUNG
   RUNG wire#w1
      Move(in := #MixingSpeed, out1 => #MixingSpeedPV)
   END_RUNG
   // the same network as SCL:
   IF #Running AND #MixingStarted THEN
       #WaterInletValve := TRUE;
       #MixerCmd := TRUE;
       #MixingSpeedPV := #MixingSpeed;
   END_IF;
END_REGION

REGION Network 6: Output Off
   RUNG wire#powerrail
      I_Contact( #Running )
      wire#w1
      R_Coil( #WaterInletValve )
   END_RUNG
   RUNG wire#w1
      R_Coil( #MixerCmd )
   END_RUNG
   RUNG wire#w1
      Move(in := 0.0, out1 => #MixingSpeedPV)
   END_RUNG
   // the same network as SCL:
   IF NOT #Running THEN
       #WaterInletValve := FALSE;
       #MixerCmd := FALSE;
       #MixingSpeedPV := 0.0;
   END_IF;
END_REGION

REGION Network 7: Event Status
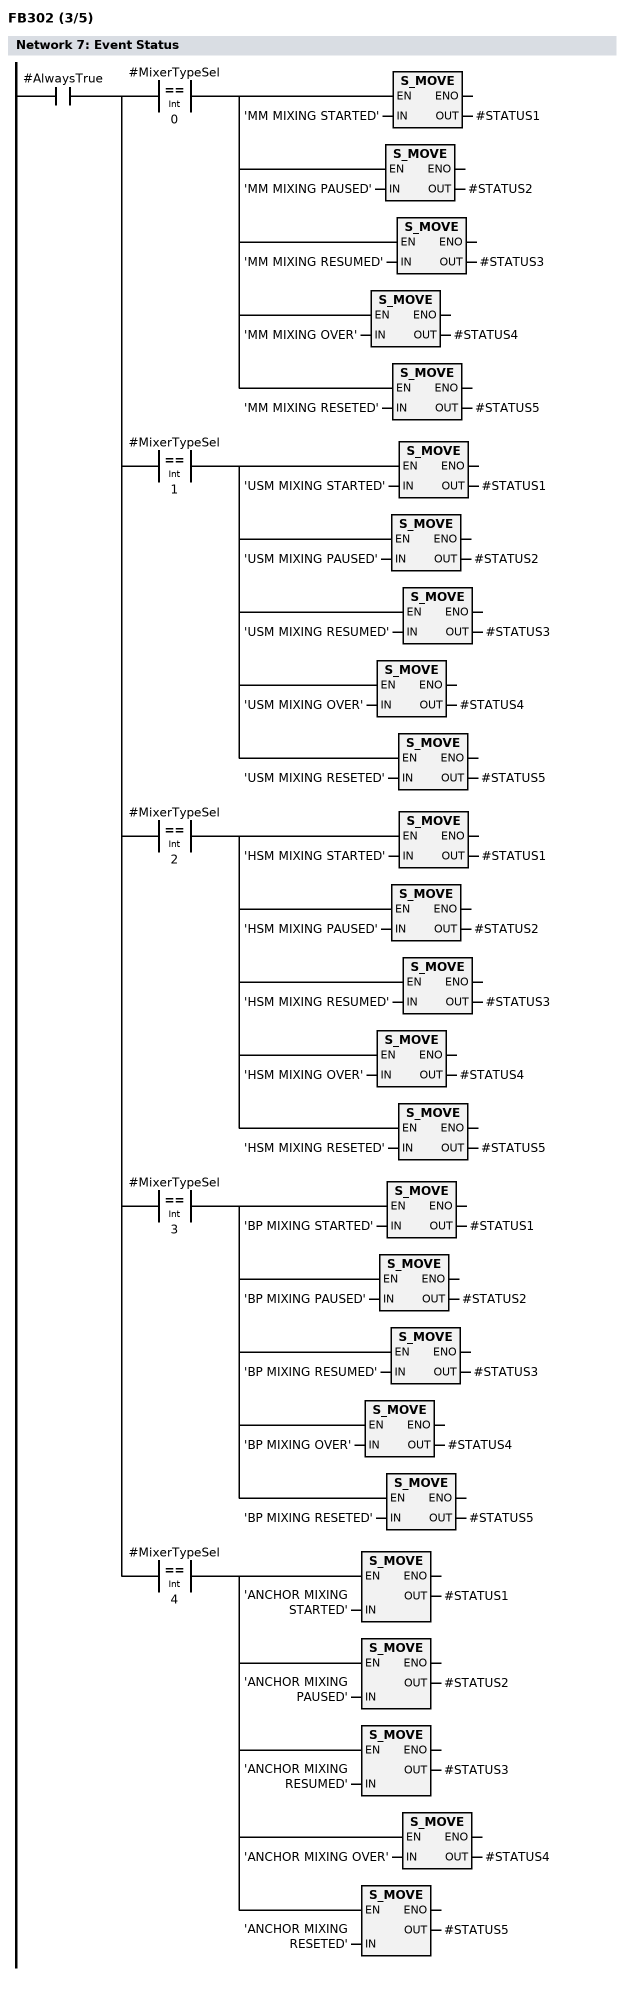
   RUNG wire#powerrail
      Contact( #AlwaysTrue )
      wire#w1
      { S7_Templates := "SrcType := Int" } EQ_Contact(in1 := #MixerTypeSel, in2 := 0)
      wire#w2
      S_Move(in := 'MM MIXING STARTED', out => #STATUS1)
   END_RUNG
   RUNG wire#w2
      S_Move(in := 'MM MIXING PAUSED', out => #STATUS2)
   END_RUNG
   RUNG wire#w2
      S_Move(in := 'MM MIXING RESUMED', out => #STATUS3)
   END_RUNG
   RUNG wire#w2
      S_Move(in := 'MM MIXING OVER', out => #STATUS4)
   END_RUNG
   RUNG wire#w2
      S_Move(in := 'MM MIXING RESETED', out => #STATUS5)
   END_RUNG
   RUNG wire#w1
      { S7_Templates := "SrcType := Int" } EQ_Contact(in1 := #MixerTypeSel, in2 := 1)
      wire#w3
      S_Move(in := 'USM MIXING STARTED', out => #STATUS1)
   END_RUNG
   RUNG wire#w3
      S_Move(in := 'USM MIXING PAUSED', out => #STATUS2)
   END_RUNG
   RUNG wire#w3
      S_Move(in := 'USM MIXING RESUMED', out => #STATUS3)
   END_RUNG
   RUNG wire#w3
      S_Move(in := 'USM MIXING OVER', out => #STATUS4)
   END_RUNG
   RUNG wire#w3
      S_Move(in := 'USM MIXING RESETED', out => #STATUS5)
   END_RUNG
   RUNG wire#w1
      { S7_Templates := "SrcType := Int" } EQ_Contact(in1 := #MixerTypeSel, in2 := 2)
      wire#w4
      S_Move(in := 'HSM MIXING STARTED', out => #STATUS1)
   END_RUNG
   RUNG wire#w4
      S_Move(in := 'HSM MIXING PAUSED', out => #STATUS2)
   END_RUNG
   RUNG wire#w4
      S_Move(in := 'HSM MIXING RESUMED', out => #STATUS3)
   END_RUNG
   RUNG wire#w4
      S_Move(in := 'HSM MIXING OVER', out => #STATUS4)
   END_RUNG
   RUNG wire#w4
      S_Move(in := 'HSM MIXING RESETED', out => #STATUS5)
   END_RUNG
   RUNG wire#w1
      { S7_Templates := "SrcType := Int" } EQ_Contact(in1 := #MixerTypeSel, in2 := 3)
      wire#w5
      S_Move(in := 'BP MIXING STARTED', out => #STATUS1)
   END_RUNG
   RUNG wire#w5
      S_Move(in := 'BP MIXING PAUSED', out => #STATUS2)
   END_RUNG
   RUNG wire#w5
      S_Move(in := 'BP MIXING RESUMED', out => #STATUS3)
   END_RUNG
   RUNG wire#w5
      S_Move(in := 'BP MIXING OVER', out => #STATUS4)
   END_RUNG
   RUNG wire#w5
      S_Move(in := 'BP MIXING RESETED', out => #STATUS5)
   END_RUNG
   RUNG wire#w1
      { S7_Templates := "SrcType := Int" } EQ_Contact(in1 := #MixerTypeSel, in2 := 4)
      wire#w6
      S_Move(in := 'ANCHOR MIXING STARTED', out => #STATUS1)
   END_RUNG
   RUNG wire#w6
      S_Move(in := 'ANCHOR MIXING PAUSED', out => #STATUS2)
   END_RUNG
   RUNG wire#w6
      S_Move(in := 'ANCHOR MIXING RESUMED', out => #STATUS3)
   END_RUNG
   RUNG wire#w6
      S_Move(in := 'ANCHOR MIXING OVER', out => #STATUS4)
   END_RUNG
   RUNG wire#w6
      S_Move(in := 'ANCHOR MIXING RESETED', out => #STATUS5)
   END_RUNG
   // the same network as SCL:
   IF #AlwaysTrue AND (#MixerTypeSel = 0) THEN
       #STATUS1 := 'MM MIXING STARTED';
       #STATUS2 := 'MM MIXING PAUSED';
       #STATUS3 := 'MM MIXING RESUMED';
       #STATUS4 := 'MM MIXING OVER';
       #STATUS5 := 'MM MIXING RESETED';
   END_IF;
   IF #AlwaysTrue AND (#MixerTypeSel = 1) THEN
       #STATUS1 := 'USM MIXING STARTED';
       #STATUS2 := 'USM MIXING PAUSED';
       #STATUS3 := 'USM MIXING RESUMED';
       #STATUS4 := 'USM MIXING OVER';
       #STATUS5 := 'USM MIXING RESETED';
   END_IF;
   IF #AlwaysTrue AND (#MixerTypeSel = 2) THEN
       #STATUS1 := 'HSM MIXING STARTED';
       #STATUS2 := 'HSM MIXING PAUSED';
       #STATUS3 := 'HSM MIXING RESUMED';
       #STATUS4 := 'HSM MIXING OVER';
       #STATUS5 := 'HSM MIXING RESETED';
   END_IF;
   IF #AlwaysTrue AND (#MixerTypeSel = 3) THEN
       #STATUS1 := 'BP MIXING STARTED';
       #STATUS2 := 'BP MIXING PAUSED';
       #STATUS3 := 'BP MIXING RESUMED';
       #STATUS4 := 'BP MIXING OVER';
       #STATUS5 := 'BP MIXING RESETED';
   END_IF;
   IF #AlwaysTrue AND (#MixerTypeSel = 4) THEN
       #STATUS1 := 'ANCHOR MIXING STARTED';
       #STATUS2 := 'ANCHOR MIXING PAUSED';
       #STATUS3 := 'ANCHOR MIXING RESUMED';
       #STATUS4 := 'ANCHOR MIXING OVER';
       #STATUS5 := 'ANCHOR MIXING RESETED';
   END_IF;
END_REGION

REGION Network 8: Print Logic
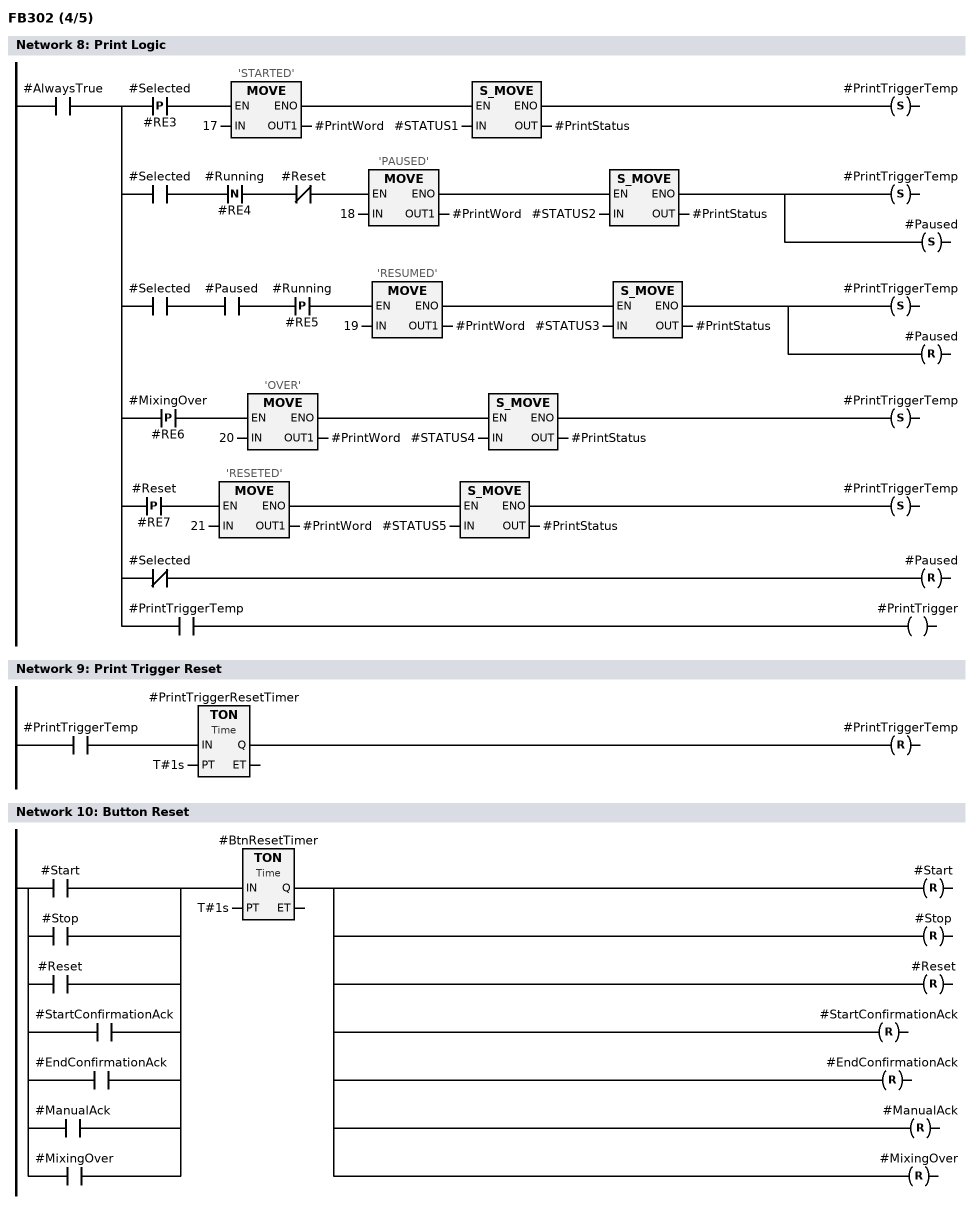
   RUNG wire#powerrail
      Contact( #AlwaysTrue )
      wire#w1
      P_Contact(operand := #Selected, bit := #RE3)
      { S7_GenerateENO := "TRUE" } Move(in := 17, out1 => #PrintWord)   // 'STARTED'
      S_Move(in := #STATUS1, out => #PrintStatus)
      S_Coil( #PrintTriggerTemp )
   END_RUNG
   RUNG wire#w1
      Contact( #Selected )
      N_Contact(operand := #Running, bit := #RE4)
      I_Contact( #Reset )
      { S7_GenerateENO := "TRUE" } Move(in := 18, out1 => #PrintWord)   // 'PAUSED'
      S_Move(in := #STATUS2, out => #PrintStatus)
      wire#w2
      S_Coil( #PrintTriggerTemp )
   END_RUNG
   RUNG wire#w2
      S_Coil( #Paused )
   END_RUNG
   RUNG wire#w1
      Contact( #Selected )
      Contact( #Paused )
      P_Contact(operand := #Running, bit := #RE5)
      { S7_GenerateENO := "TRUE" } Move(in := 19, out1 => #PrintWord)   // 'RESUMED'
      S_Move(in := #STATUS3, out => #PrintStatus)
      wire#w3
      S_Coil( #PrintTriggerTemp )
   END_RUNG
   RUNG wire#w3
      R_Coil( #Paused )
   END_RUNG
   RUNG wire#w1
      P_Contact(operand := #MixingOver, bit := #RE6)
      { S7_GenerateENO := "TRUE" } Move(in := 20, out1 => #PrintWord)   // 'OVER'
      S_Move(in := #STATUS4, out => #PrintStatus)
      S_Coil( #PrintTriggerTemp )
   END_RUNG
   RUNG wire#w1
      P_Contact(operand := #Reset, bit := #RE7)
      { S7_GenerateENO := "TRUE" } Move(in := 21, out1 => #PrintWord)   // 'RESETED'
      S_Move(in := #STATUS5, out => #PrintStatus)
      S_Coil( #PrintTriggerTemp )
   END_RUNG
   RUNG wire#w1
      I_Contact( #Selected )
      R_Coil( #Paused )
   END_RUNG
   RUNG wire#w1
      Contact( #PrintTriggerTemp )
      Coil( #PrintTrigger )
   END_RUNG
   // the same network as SCL:
   // ENO of a box is taken as its EN; it also drops when the box reports an error
   #_w1 := #AlwaysTrue AND #Selected AND NOT #RE3;   // rising edge of #Selected
   #RE3 := #Selected;
   IF #_w1 THEN
       #PrintWord := 17;   // 'STARTED'
       #PrintStatus := #STATUS1;
       #PrintTriggerTemp := TRUE;
   END_IF;
   #_w2 := #AlwaysTrue AND #Selected AND NOT #Running AND #RE4;   // falling edge of #Running
   #RE4 := #Running;
   IF #_w2 AND NOT #Reset THEN
       #PrintWord := 18;   // 'PAUSED'
       #PrintStatus := #STATUS2;
       #PrintTriggerTemp := TRUE;
       #Paused := TRUE;
   END_IF;
   #_w3 := #AlwaysTrue AND #Selected AND #Paused AND #Running AND NOT #RE5;   // rising edge of #Running
   #RE5 := #Running;
   IF #_w3 THEN
       #PrintWord := 19;   // 'RESUMED'
       #PrintStatus := #STATUS3;
       #PrintTriggerTemp := TRUE;
       #Paused := FALSE;
   END_IF;
   #_w4 := #AlwaysTrue AND #MixingOver AND NOT #RE6;   // rising edge of #MixingOver
   #RE6 := #MixingOver;
   IF #_w4 THEN
       #PrintWord := 20;   // 'OVER'
       #PrintStatus := #STATUS4;
       #PrintTriggerTemp := TRUE;
   END_IF;
   #_w5 := #AlwaysTrue AND #Reset AND NOT #RE7;   // rising edge of #Reset
   #RE7 := #Reset;
   IF #_w5 THEN
       #PrintWord := 21;   // 'RESETED'
       #PrintStatus := #STATUS5;
       #PrintTriggerTemp := TRUE;
   END_IF;
   IF #AlwaysTrue AND NOT #Selected THEN #Paused := FALSE; END_IF;
   #PrintTrigger := #AlwaysTrue AND #PrintTriggerTemp;
END_REGION

REGION Network 9: Print Trigger Reset
   RUNG wire#powerrail
      Contact( #PrintTriggerTemp )
      { S7_Templates := "time_type := Time" } #PrintTriggerResetTimer.TON(pt := T#1s, et =>)
      R_Coil( #PrintTriggerTemp )
   END_RUNG
   // the same network as SCL:
   #PrintTriggerResetTimer(IN := #PrintTriggerTemp, PT := T#1s);   // TON
   IF #PrintTriggerResetTimer.Q THEN #PrintTriggerTemp := FALSE; END_IF;
END_REGION

REGION Network 10: Button Reset
   RUNG wire#powerrail
      Contact( #Start )
      wire#w1
      { S7_Templates := "time_type := Time" } #BtnResetTimer.TON(pt := T#1s, et =>)
      wire#w2
      R_Coil( #Start )
   END_RUNG
   RUNG wire#powerrail
      Contact( #Stop )
   END_RUNG wire#w1
   RUNG wire#powerrail
      Contact( #Reset )
   END_RUNG wire#w1
   RUNG wire#powerrail
      Contact( #StartConfirmationAck )
   END_RUNG wire#w1
   RUNG wire#powerrail
      Contact( #EndConfirmationAck )
   END_RUNG wire#w1
   RUNG wire#powerrail
      Contact( #ManualAck )
   END_RUNG wire#w1
   RUNG wire#powerrail
      Contact( #MixingOver )
   END_RUNG wire#w1
   RUNG wire#w2
      R_Coil( #Stop )
   END_RUNG
   RUNG wire#w2
      R_Coil( #Reset )
   END_RUNG
   RUNG wire#w2
      R_Coil( #StartConfirmationAck )
   END_RUNG
   RUNG wire#w2
      R_Coil( #EndConfirmationAck )
   END_RUNG
   RUNG wire#w2
      R_Coil( #ManualAck )
   END_RUNG
   RUNG wire#w2
      R_Coil( #MixingOver )
   END_RUNG
   // the same network as SCL:
   #BtnResetTimer(IN := #Start OR #Stop OR #Reset OR #StartConfirmationAck OR #EndConfirmationAck OR #ManualAck OR #MixingOver,   // TON
                  PT := T#1s);
   IF #BtnResetTimer.Q THEN
       #Start := FALSE;
       #Stop := FALSE;
       #Reset := FALSE;
       #StartConfirmationAck := FALSE;
       #EndConfirmationAck := FALSE;
       #ManualAck := FALSE;
       #MixingOver := FALSE;
   END_IF;
END_REGION

REGION Network 11: Reset
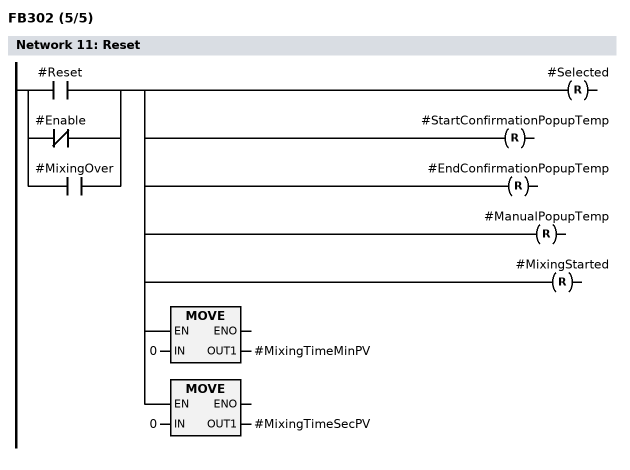
   RUNG wire#powerrail
      Contact( #Reset )
      wire#w1
      R_Coil( #Selected )
   END_RUNG
   RUNG wire#powerrail
      I_Contact( #Enable )
   END_RUNG wire#w1
   RUNG wire#powerrail
      Contact( #MixingOver )
   END_RUNG wire#w1
   RUNG wire#w1
      R_Coil( #StartConfirmationPopupTemp )
   END_RUNG
   RUNG wire#w1
      R_Coil( #EndConfirmationPopupTemp )
   END_RUNG
   RUNG wire#w1
      R_Coil( #ManualPopupTemp )
   END_RUNG
   RUNG wire#w1
      R_Coil( #MixingStarted )
   END_RUNG
   RUNG wire#w1
      { S7_GenerateENO := "TRUE" } Move(in := 0, out1 => #MixingTimeMinPV)
   END_RUNG
   RUNG wire#w1
      { S7_GenerateENO := "TRUE" } Move(in := 0, out1 => #MixingTimeSecPV)
   END_RUNG
   // the same network as SCL:
   IF #Reset OR NOT #Enable OR #MixingOver THEN
       #Selected := FALSE;
       #StartConfirmationPopupTemp := FALSE;
       #EndConfirmationPopupTemp := FALSE;
       #ManualPopupTemp := FALSE;
       #MixingStarted := FALSE;
       #MixingTimeMinPV := 0;
       #MixingTimeSecPV := 0;
   END_IF;
END_REGION
END_FUNCTION_BLOCK

FUNCTION_BLOCK "FB310"   // FB310, LAD
TITLE = FB310
{ S7_Optimized_Access := 'TRUE' }
AUTHOR : PRECISE
FAMILY : PRECISE
// RAW MATERIAL ADDITION 
// 0-MANUAL/1-SUCTION/2-LIQUID DRUM
// stored: AutoNumber false, MemoryReserve 100, SetENOAutomatically false
   VAR_INPUT
      Enable : Bool;
      Disable : Bool;
      Fault : Bool;
      SecPulse : Bool;
      AlwaysTrue : Bool;
      StartConfirmationPopupSel : Bool;   // StartConfirmationPopupSel: 0-NO/1-YES
      EndConfirmationPopupSel : Bool;   // EndConfirmationPopupSel: 0-NO/1-YES
      RMAddTypeSel : Int;   // RMAddTypeSel: 0-Manual/1-Suction/2-Liquid Drum
      RMTypeSel : Int := 1;   // RM Type Sel: Graules or Flakes -0/FinePowder-1
      WeightBasedSel : Bool;   // Weight Based Sel: 0-NO/1-YES
      AdditionMethodSel : Bool;   // Addition Method : 0-Add In Weight/1-Loss In Weight
      RMAddPopupSel : Bool;   // RM Add Popup Sel: 0-NO/1-YES
      SetRMNo : Int := 1;
      "SetVacuum/SetPressure" : Real := -300.0;   // SetVauum - For unit "mmHg" / SetPressure - For unit "bar"
      SetQuantity : Real := 10.0;   // Weight Based Sel: 1-YES
      SetSpeed : Real := 50.0;
      "ActualVacuum/ActualPressure" : Real;   // ActualVauum - For unit "mmHg" / ActualPressure - For unit "bar"
      ActualQuantity : Real;   // Collecting Vessel Weight
      ActualQuantityRMVessel : Real;   // Transffering Vessel Weight
      "VacuumTol/PressureTol" : Real := 10.0;   // VacuumTol - For unit "mmHg" / PressureTol - For unit "bar"
      DelaytoSettleMaterial : Int := 5;
      InflightQuantitySuction : Real;
      InflightQuantityLiqDrum : Real;
      DelaytoStartPump : Int := 3;
   END_VAR
   VAR_OUTPUT
      VacuumInValve : Bool;
      VacuumLineValves : Bool;
      SuctionInValve : Bool;
      VacuumPumpCmd : Bool;
      LineValves : Bool;
      PumpCmd : Bool;
      StartConfirmationPopup : Bool;   // For Start Confirmation Popup Selection: Yes
      EndConfirmationPopup : Bool;   // For End Confirmation Popup Selection: Yes
      DelaytoSettleMaterialPopup : Bool;   // "WAITING FOR MATERIAL TO SETTLE"
      RMAddPopup : Bool;   // For RMAddPopupSel: 1-YES
      RMAddPopupManual : Bool;   // For RMAddPopupSel: 1-YES
      ActualSpeed : Real;
      VisibleRM1 : Bool;
      VisibleRM2 : Bool;
      VisibleRM3 : Bool;
      VisibleRM4 : Bool;
      VisibleRM5 : Bool;
      VisibleRM6 : Bool;
      VisibleRM7 : Bool;
      VisibleRM8 : Bool;
      VisibleRM9 : Bool;
      VisibleRM10 : Bool;
      PrintTrigger : Bool;
      PrintWord : Int;
      PrintStatus : String[50];
   END_VAR
   VAR_IN_OUT
      Start : Bool;
      Stop : Bool;
      Reset : Bool;
      StartConfirmationAck : Bool;   // For Start Confirmation Popup Selection: Yes
      EndConfirmationAck : Bool;   // For End Confirmation Popup Selection: Yes
      SpareBtn1 : Bool;
      SpareBtn2 : Bool;
      Running : Bool;
      Selected : Bool;
      Paused : Bool;
      StartConfirmationPopupTemp : Bool;   // For Start Confirmation Popup Selection: Yes
      EndConfirmationPopupTemp : Bool;   // For End Confirmation Popup Selection: Yes
      RMAddPopupTemp : Bool;   // For RMAddPopupSel: 1-YES
      RMAddStarted : Bool;
      RMAddOver : Bool;
      ActualSetQuantityCalc : Real;   // For WeightBaseSel: 1-YES
      ActualSetQuantity : Real;   // For WeightBaseSel: 1-YES
      RMAddAck1 : Bool;   // For RMAddPopupSel: 1-YES
      RMAddAck2 : Bool;   // For RMAddPopupSel: 1-YES
      RMAddAck3 : Bool;   // For RMAddPopupSel: 1-YES
      RMAddAck4 : Bool;   // For RMAddPopupSel: 1-YES
      RMAddAck5 : Bool;   // For RMAddPopupSel: 1-YES
      RMAddAck6 : Bool;   // For RMAddPopupSel: 1-YES
      RMAddAck7 : Bool;   // For RMAddPopupSel: 1-YES
      RMAddAck8 : Bool;   // For RMAddPopupSel: 1-YES
      RMAddAck9 : Bool;   // For RMAddPopupSel: 1-YES
      RMAddAck10 : Bool;   // For RMAddPopupSel: 1-YES
   END_VAR
   VAR
      PrintTriggerTemp : Bool;
      RE1 : Bool;
      RE2 : Bool;
      RE3 : Bool;
      RE4 : Bool;
      RE5 : Bool;
      RE6 : Bool;
      RE7 : Bool;
      RE8 : Bool;
      RE9 : Bool;
      RE10 : Bool;
      RE11 : Bool;
      PrintTriggerResetTimer { S7_SetPoint := 'True'} : TON_TIME;
      BtnResetTimer { S7_SetPoint := 'True'} : TON_TIME;
   END_VAR
   VAR RETAIN
      NameRM1 : String[100];
   END_VAR
   VAR
      NameRM2 : String[100];
      NameRM3 : String[100];
      NameRM4 : String[100];
      NameRM5 : String[100];
      NameRM6 : String[100];
      NameRM7 : String[100];
      NameRM8 : String[100];
      NameRM9 : String[100];
      NameRM10 : String[100];
      Manual { S7_SetPoint := 'True'} : "FB307";
      Suction { S7_SetPoint := 'True'} : "FB308";
      LiqDrum { S7_SetPoint := 'True'} : "FB309";
   END_VAR
   VAR_TEMP
      STATUS1 : String[40];
      STATUS2 : String[40];
      STATUS3 : String[40];
      STATUS4 : String[40];
      STATUS5 : String[40];
      Blank : String[40];
   END_VAR
   VAR_TEMP   // added for the SCL form of the ladder/FBD networks
      _w1 : Bool;
      _w2 : Bool;
      _w3 : Bool;
      _w4 : Bool;
      _w5 : Bool;
      _w6 : Bool;
   END_VAR
BEGIN

REGION Network 1: Running
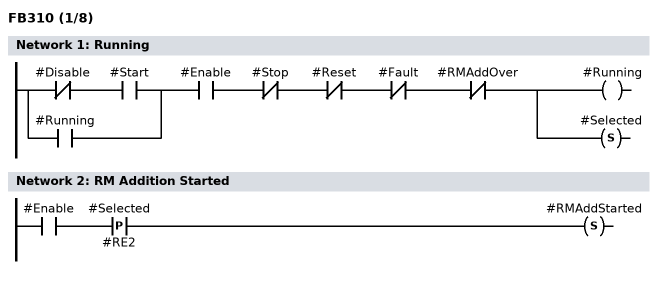
   RUNG wire#powerrail
      I_Contact( #Disable )
      Contact( #Start )
      wire#w1
      Contact( #Enable )
      I_Contact( #Stop )
      I_Contact( #Reset )
      I_Contact( #Fault )
      I_Contact( #RMAddOver )
      wire#w2
      Coil( #Running )
   END_RUNG
   RUNG wire#powerrail
      Contact( #Running )
   END_RUNG wire#w1
   RUNG wire#w2
      S_Coil( #Selected )
   END_RUNG
   // the same network as SCL:
   #Running := ((NOT #Disable AND #Start) OR #Running) AND #Enable AND NOT #Stop AND NOT #Reset AND NOT #Fault AND NOT #RMAddOver;
   IF #Running THEN #Selected := TRUE; END_IF;
END_REGION

REGION Network 2: RM Addition Started
   RUNG wire#powerrail
      Contact( #Enable )
      P_Contact(operand := #Selected, bit := #RE2)
      S_Coil( #RMAddStarted )
   END_RUNG
   // the same network as SCL:
   #_w1 := #Enable AND #Selected AND NOT #RE2;   // rising edge of #Selected
   #RE2 := #Selected;
   IF #_w1 THEN #RMAddStarted := TRUE; END_IF;
END_REGION

REGION Network 3: RM Addition Parameters
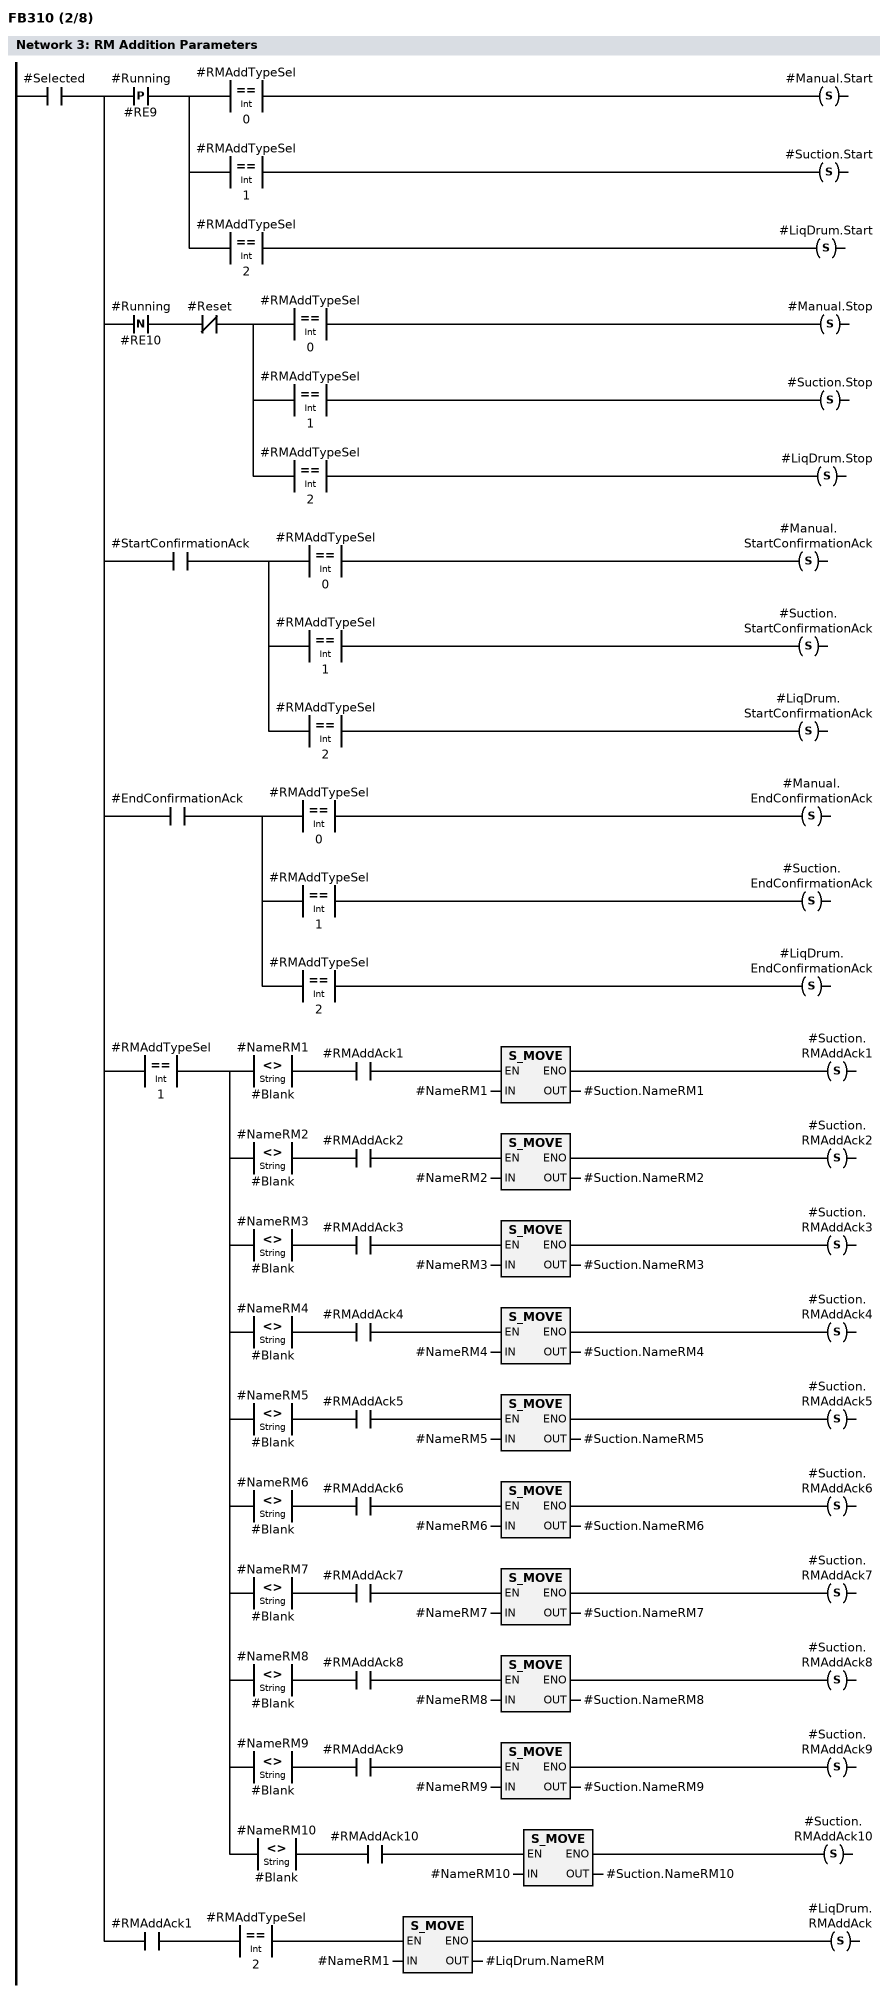
   RUNG wire#powerrail
      Contact( #Selected )
      wire#w1
      P_Contact(operand := #Running, bit := #RE9)
      wire#w2
      { S7_Templates := "SrcType := Int" } EQ_Contact(in1 := #RMAddTypeSel, in2 := 0)
      S_Coil( #Manual.Start )
   END_RUNG
   RUNG wire#w2
      { S7_Templates := "SrcType := Int" } EQ_Contact(in1 := #RMAddTypeSel, in2 := 1)
      S_Coil( #Suction.Start )
   END_RUNG
   RUNG wire#w2
      { S7_Templates := "SrcType := Int" } EQ_Contact(in1 := #RMAddTypeSel, in2 := 2)
      S_Coil( #LiqDrum.Start )
   END_RUNG
   RUNG wire#w1
      N_Contact(operand := #Running, bit := #RE10)
      I_Contact( #Reset )
      wire#w3
      { S7_Templates := "SrcType := Int" } EQ_Contact(in1 := #RMAddTypeSel, in2 := 0)
      S_Coil( #Manual.Stop )
   END_RUNG
   RUNG wire#w3
      { S7_Templates := "SrcType := Int" } EQ_Contact(in1 := #RMAddTypeSel, in2 := 1)
      S_Coil( #Suction.Stop )
   END_RUNG
   RUNG wire#w3
      { S7_Templates := "SrcType := Int" } EQ_Contact(in1 := #RMAddTypeSel, in2 := 2)
      S_Coil( #LiqDrum.Stop )
   END_RUNG
   RUNG wire#w1
      Contact( #StartConfirmationAck )
      wire#w4
      { S7_Templates := "SrcType := Int" } EQ_Contact(in1 := #RMAddTypeSel, in2 := 0)
      S_Coil( #Manual.StartConfirmationAck )
   END_RUNG
   RUNG wire#w4
      { S7_Templates := "SrcType := Int" } EQ_Contact(in1 := #RMAddTypeSel, in2 := 1)
      S_Coil( #Suction.StartConfirmationAck )
   END_RUNG
   RUNG wire#w4
      { S7_Templates := "SrcType := Int" } EQ_Contact(in1 := #RMAddTypeSel, in2 := 2)
      S_Coil( #LiqDrum.StartConfirmationAck )
   END_RUNG
   RUNG wire#w1
      Contact( #EndConfirmationAck )
      wire#w5
      { S7_Templates := "SrcType := Int" } EQ_Contact(in1 := #RMAddTypeSel, in2 := 0)
      S_Coil( #Manual.EndConfirmationAck )
   END_RUNG
   RUNG wire#w5
      { S7_Templates := "SrcType := Int" } EQ_Contact(in1 := #RMAddTypeSel, in2 := 1)
      S_Coil( #Suction.EndConfirmationAck )
   END_RUNG
   RUNG wire#w5
      { S7_Templates := "SrcType := Int" } EQ_Contact(in1 := #RMAddTypeSel, in2 := 2)
      S_Coil( #LiqDrum.EndConfirmationAck )
   END_RUNG
   RUNG wire#w1
      { S7_Templates := "SrcType := Int" } EQ_Contact(in1 := #RMAddTypeSel, in2 := 1)
      wire#w6
      { S7_Templates := "SrcType := String" } NE_Contact(in1 := #NameRM1, in2 := #Blank)
      Contact( #RMAddAck1 )
      S_Move(in := #NameRM1, out => #Suction.NameRM1)
      S_Coil( #Suction.RMAddAck1 )
   END_RUNG
   RUNG wire#w6
      { S7_Templates := "SrcType := String" } NE_Contact(in1 := #NameRM2, in2 := #Blank)
      Contact( #RMAddAck2 )
      S_Move(in := #NameRM2, out => #Suction.NameRM2)
      S_Coil( #Suction.RMAddAck2 )
   END_RUNG
   RUNG wire#w6
      { S7_Templates := "SrcType := String" } NE_Contact(in1 := #NameRM3, in2 := #Blank)
      Contact( #RMAddAck3 )
      S_Move(in := #NameRM3, out => #Suction.NameRM3)
      S_Coil( #Suction.RMAddAck3 )
   END_RUNG
   RUNG wire#w6
      { S7_Templates := "SrcType := String" } NE_Contact(in1 := #NameRM4, in2 := #Blank)
      Contact( #RMAddAck4 )
      S_Move(in := #NameRM4, out => #Suction.NameRM4)
      S_Coil( #Suction.RMAddAck4 )
   END_RUNG
   RUNG wire#w6
      { S7_Templates := "SrcType := String" } NE_Contact(in1 := #NameRM5, in2 := #Blank)
      Contact( #RMAddAck5 )
      S_Move(in := #NameRM5, out => #Suction.NameRM5)
      S_Coil( #Suction.RMAddAck5 )
   END_RUNG
   RUNG wire#w6
      { S7_Templates := "SrcType := String" } NE_Contact(in1 := #NameRM6, in2 := #Blank)
      Contact( #RMAddAck6 )
      S_Move(in := #NameRM6, out => #Suction.NameRM6)
      S_Coil( #Suction.RMAddAck6 )
   END_RUNG
   RUNG wire#w6
      { S7_Templates := "SrcType := String" } NE_Contact(in1 := #NameRM7, in2 := #Blank)
      Contact( #RMAddAck7 )
      S_Move(in := #NameRM7, out => #Suction.NameRM7)
      S_Coil( #Suction.RMAddAck7 )
   END_RUNG
   RUNG wire#w6
      { S7_Templates := "SrcType := String" } NE_Contact(in1 := #NameRM8, in2 := #Blank)
      Contact( #RMAddAck8 )
      S_Move(in := #NameRM8, out => #Suction.NameRM8)
      S_Coil( #Suction.RMAddAck8 )
   END_RUNG
   RUNG wire#w6
      { S7_Templates := "SrcType := String" } NE_Contact(in1 := #NameRM9, in2 := #Blank)
      Contact( #RMAddAck9 )
      S_Move(in := #NameRM9, out => #Suction.NameRM9)
      S_Coil( #Suction.RMAddAck9 )
   END_RUNG
   RUNG wire#w6
      { S7_Templates := "SrcType := String" } NE_Contact(in1 := #NameRM10, in2 := #Blank)
      Contact( #RMAddAck10 )
      S_Move(in := #NameRM10, out => #Suction.NameRM10)
      S_Coil( #Suction.RMAddAck10 )
   END_RUNG
   RUNG wire#w1
      Contact( #RMAddAck1 )
      { S7_Templates := "SrcType := Int" } EQ_Contact(in1 := #RMAddTypeSel, in2 := 2)
      S_Move(in := #NameRM1, out => #LiqDrum.NameRM)
      S_Coil( #LiqDrum.RMAddAck )
   END_RUNG
   // the same network as SCL:
   #_w1 := #Selected AND #Running AND NOT #RE9;   // rising edge of #Running
   #RE9 := #Running;
   IF #_w1 AND (#RMAddTypeSel = 0) THEN #Manual.Start := TRUE; END_IF;
   IF #_w1 AND (#RMAddTypeSel = 1) THEN #Suction.Start := TRUE; END_IF;
   IF #_w1 AND (#RMAddTypeSel = 2) THEN #LiqDrum.Start := TRUE; END_IF;
   #_w2 := #Selected AND NOT #Running AND #RE10;   // falling edge of #Running
   #RE10 := #Running;
   #_w3 := #_w2 AND NOT #Reset;
   IF #_w3 AND (#RMAddTypeSel = 0) THEN #Manual.Stop := TRUE; END_IF;
   IF #_w3 AND (#RMAddTypeSel = 1) THEN #Suction.Stop := TRUE; END_IF;
   IF #_w3 AND (#RMAddTypeSel = 2) THEN #LiqDrum.Stop := TRUE; END_IF;
   #_w4 := #Selected AND #StartConfirmationAck;
   IF #_w4 AND (#RMAddTypeSel = 0) THEN #Manual.StartConfirmationAck := TRUE; END_IF;
   IF #_w4 AND (#RMAddTypeSel = 1) THEN #Suction.StartConfirmationAck := TRUE; END_IF;
   IF #_w4 AND (#RMAddTypeSel = 2) THEN #LiqDrum.StartConfirmationAck := TRUE; END_IF;
   #_w5 := #Selected AND #EndConfirmationAck;
   IF #_w5 AND (#RMAddTypeSel = 0) THEN #Manual.EndConfirmationAck := TRUE; END_IF;
   IF #_w5 AND (#RMAddTypeSel = 1) THEN #Suction.EndConfirmationAck := TRUE; END_IF;
   IF #_w5 AND (#RMAddTypeSel = 2) THEN #LiqDrum.EndConfirmationAck := TRUE; END_IF;
   #_w6 := #Selected AND (#RMAddTypeSel = 1);
   IF #_w6 AND (#NameRM1 <> #Blank) AND #RMAddAck1 THEN
       #Suction.NameRM1 := #NameRM1;
       #Suction.RMAddAck1 := TRUE;
   END_IF;
   IF #_w6 AND (#NameRM2 <> #Blank) AND #RMAddAck2 THEN
       #Suction.NameRM2 := #NameRM2;
       #Suction.RMAddAck2 := TRUE;
   END_IF;
   IF #_w6 AND (#NameRM3 <> #Blank) AND #RMAddAck3 THEN
       #Suction.NameRM3 := #NameRM3;
       #Suction.RMAddAck3 := TRUE;
   END_IF;
   IF #_w6 AND (#NameRM4 <> #Blank) AND #RMAddAck4 THEN
       #Suction.NameRM4 := #NameRM4;
       #Suction.RMAddAck4 := TRUE;
   END_IF;
   IF #_w6 AND (#NameRM5 <> #Blank) AND #RMAddAck5 THEN
       #Suction.NameRM5 := #NameRM5;
       #Suction.RMAddAck5 := TRUE;
   END_IF;
   IF #_w6 AND (#NameRM6 <> #Blank) AND #RMAddAck6 THEN
       #Suction.NameRM6 := #NameRM6;
       #Suction.RMAddAck6 := TRUE;
   END_IF;
   IF #_w6 AND (#NameRM7 <> #Blank) AND #RMAddAck7 THEN
       #Suction.NameRM7 := #NameRM7;
       #Suction.RMAddAck7 := TRUE;
   END_IF;
   IF #_w6 AND (#NameRM8 <> #Blank) AND #RMAddAck8 THEN
       #Suction.NameRM8 := #NameRM8;
       #Suction.RMAddAck8 := TRUE;
   END_IF;
   IF #_w6 AND (#NameRM9 <> #Blank) AND #RMAddAck9 THEN
       #Suction.NameRM9 := #NameRM9;
       #Suction.RMAddAck9 := TRUE;
   END_IF;
   IF #_w6 AND (#NameRM10 <> #Blank) AND #RMAddAck10 THEN
       #Suction.NameRM10 := #NameRM10;
       #Suction.RMAddAck10 := TRUE;
   END_IF;
   IF #Selected AND #RMAddAck1 AND (#RMAddTypeSel = 2) THEN
       #LiqDrum.NameRM := #NameRM1;
       #LiqDrum.RMAddAck := TRUE;
   END_IF;
END_REGION

REGION Network 4: RM Addition Manual
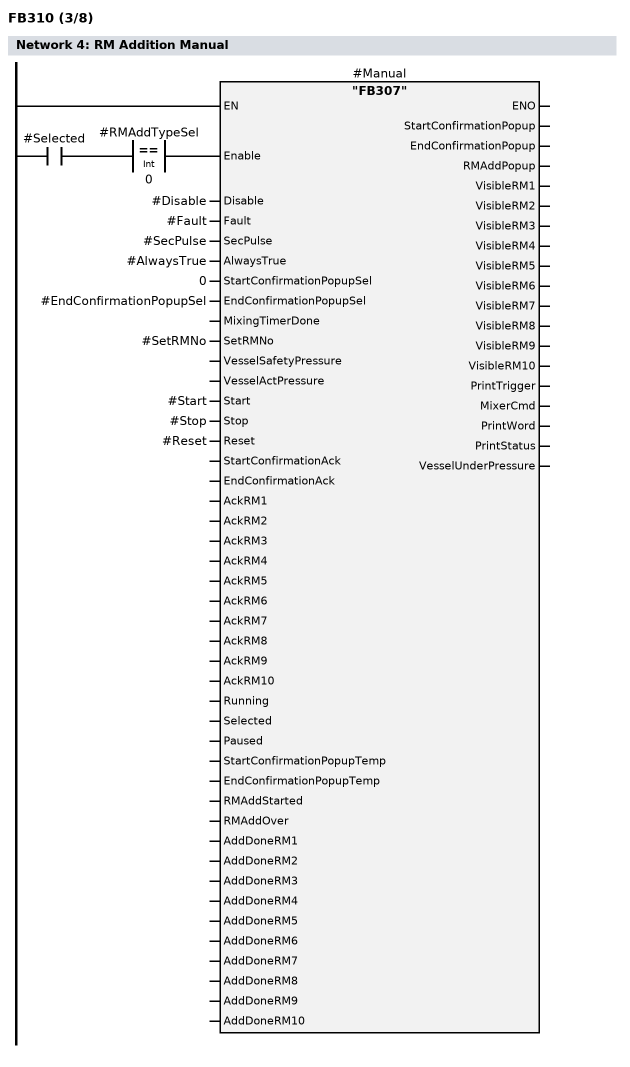
   RUNG wire#powerrail
      #Manual(Enable := wire#w1, Disable := #Disable, Fault := #Fault, SecPulse := #SecPulse, AlwaysTrue := #AlwaysTrue, StartConfirmationPopupSel := 0, EndConfirmationPopupSel := #EndConfirmationPopupSel, MixingTimerDone :=, SetRMNo := #SetRMNo, VesselSafetyPressure :=, VesselActPressure :=, Start := #Start, Stop := #Stop, Reset := #Reset, StartConfirmationAck :=, EndConfirmationAck :=, AckRM1 :=, AckRM2 :=, AckRM3 :=, AckRM4 :=, AckRM5 :=, AckRM6 :=, AckRM7 :=, AckRM8 :=, AckRM9 :=, AckRM10 :=, Running :=, Selected :=, Paused :=, StartConfirmationPopupTemp :=, EndConfirmationPopupTemp :=, RMAddStarted :=, RMAddOver :=, AddDoneRM1 :=, AddDoneRM2 :=, AddDoneRM3 :=, AddDoneRM4 :=, AddDoneRM5 :=, AddDoneRM6 :=, AddDoneRM7 :=, AddDoneRM8 :=, AddDoneRM9 :=, AddDoneRM10 :=, StartConfirmationPopup =>, EndConfirmationPopup =>, RMAddPopup =>, VisibleRM1 =>, VisibleRM2 =>, VisibleRM3 =>, VisibleRM4 =>, VisibleRM5 =>, VisibleRM6 =>, VisibleRM7 =>, VisibleRM8 =>, VisibleRM9 =>, VisibleRM10 =>, PrintTrigger =>, MixerCmd =>, PrintWord =>, PrintStatus =>, VesselUnderPressure =>)
   END_RUNG
   RUNG wire#powerrail
      Contact( #Selected )
      { S7_Templates := "SrcType := Int" } EQ_Contact(in1 := #RMAddTypeSel, in2 := 0)
   END_RUNG wire#w1
   // the same network as SCL:
   #Manual(Enable := #Selected AND (#RMAddTypeSel = 0),   // "FB307"
           Disable := #Disable,
           Fault := #Fault,
           SecPulse := #SecPulse,
           AlwaysTrue := #AlwaysTrue,
           StartConfirmationPopupSel := 0,
           EndConfirmationPopupSel := #EndConfirmationPopupSel,
           SetRMNo := #SetRMNo,
           Start := #Start,
           Stop := #Stop,
           Reset := #Reset);
END_REGION

REGION Network 5: RM Addition Suction
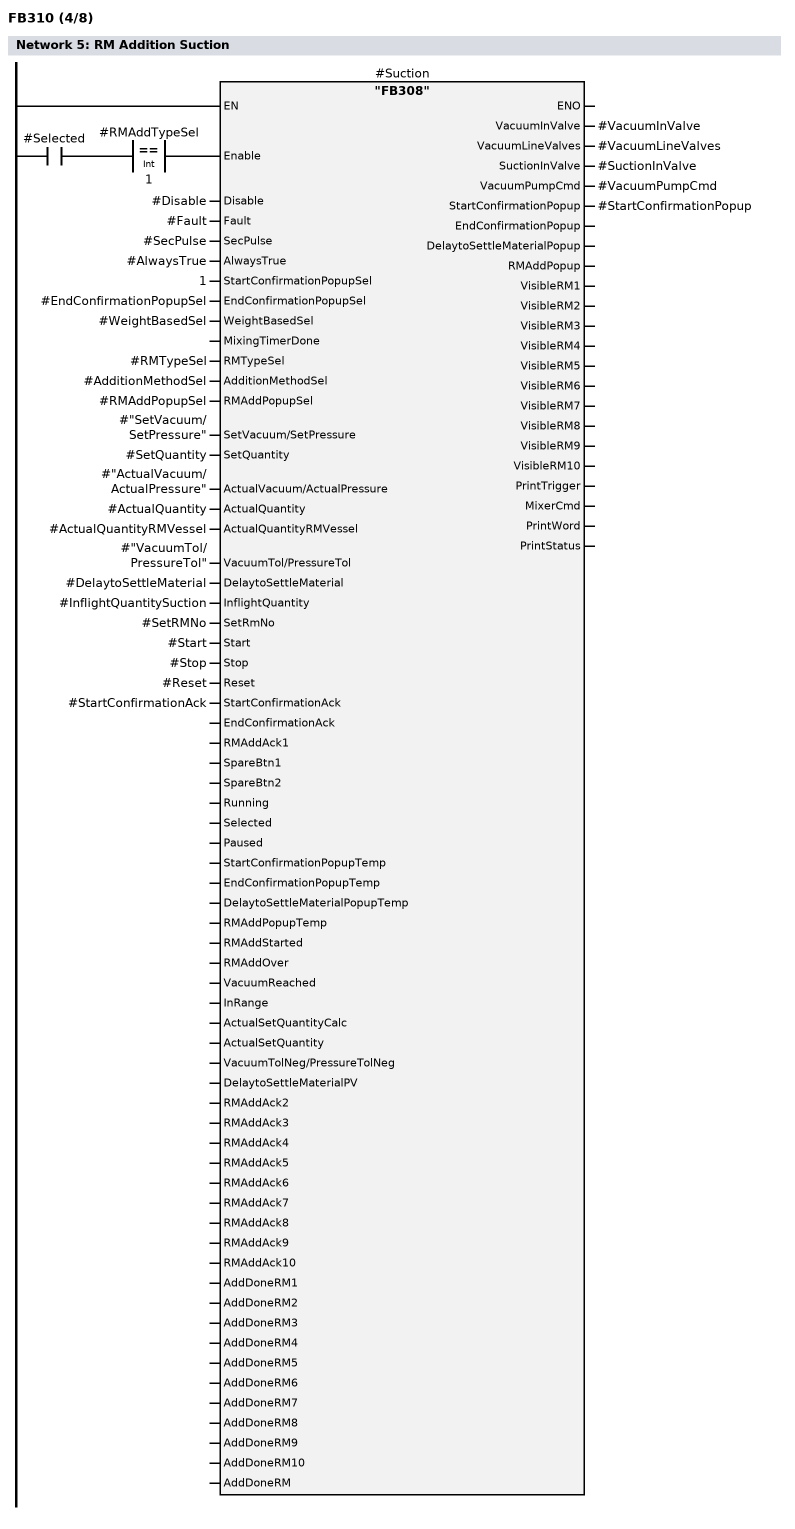
   RUNG wire#powerrail
      #Suction(Enable := wire#w1, Disable := #Disable, Fault := #Fault, SecPulse := #SecPulse, AlwaysTrue := #AlwaysTrue, StartConfirmationPopupSel := 1, EndConfirmationPopupSel := #EndConfirmationPopupSel, WeightBasedSel := #WeightBasedSel, MixingTimerDone :=, RMTypeSel := #RMTypeSel, AdditionMethodSel := #AdditionMethodSel, RMAddPopupSel := #RMAddPopupSel, "SetVacuum/SetPressure" := #"SetVacuum/SetPressure", SetQuantity := #SetQuantity, "ActualVacuum/ActualPressure" := #"ActualVacuum/ActualPressure", ActualQuantity := #ActualQuantity, ActualQuantityRMVessel := #ActualQuantityRMVessel, "VacuumTol/PressureTol" := #"VacuumTol/PressureTol", DelaytoSettleMaterial := #DelaytoSettleMaterial, InflightQuantity := #InflightQuantitySuction, SetRmNo := #SetRMNo, Start := #Start, Stop := #Stop, Reset := #Reset, StartConfirmationAck := #StartConfirmationAck, EndConfirmationAck :=, RMAddAck1 :=, SpareBtn1 :=, SpareBtn2 :=, Running :=, Selected :=, Paused :=, StartConfirmationPopupTemp :=, EndConfirmationPopupTemp :=, DelaytoSettleMaterialPopupTemp :=, RMAddPopupTemp :=, RMAddStarted :=, RMAddOver :=, VacuumReached :=, InRange :=, ActualSetQuantityCalc :=, ActualSetQuantity :=, "VacuumTolNeg/PressureTolNeg" :=, DelaytoSettleMaterialPV :=, RMAddAck2 :=, RMAddAck3 :=, RMAddAck4 :=, RMAddAck5 :=, RMAddAck6 :=, RMAddAck7 :=, RMAddAck8 :=, RMAddAck9 :=, RMAddAck10 :=, AddDoneRM1 :=, AddDoneRM2 :=, AddDoneRM3 :=, AddDoneRM4 :=, AddDoneRM5 :=, AddDoneRM6 :=, AddDoneRM7 :=, AddDoneRM8 :=, AddDoneRM9 :=, AddDoneRM10 :=, AddDoneRM :=, VacuumInValve => #VacuumInValve, VacuumLineValves => #VacuumLineValves, SuctionInValve => #SuctionInValve, VacuumPumpCmd => #VacuumPumpCmd, StartConfirmationPopup => #StartConfirmationPopup, EndConfirmationPopup =>, DelaytoSettleMaterialPopup =>, RMAddPopup =>, VisibleRM1 =>, VisibleRM2 =>, VisibleRM3 =>, VisibleRM4 =>, VisibleRM5 =>, VisibleRM6 =>, VisibleRM7 =>, VisibleRM8 =>, VisibleRM9 =>, VisibleRM10 =>, PrintTrigger =>, MixerCmd =>, PrintWord =>, PrintStatus =>)
   END_RUNG
   RUNG wire#powerrail
      Contact( #Selected )
      { S7_Templates := "SrcType := Int" } EQ_Contact(in1 := #RMAddTypeSel, in2 := 1)
   END_RUNG wire#w1
   // the same network as SCL:
   #Suction(Enable := #Selected AND (#RMAddTypeSel = 1),   // "FB308"
            Disable := #Disable,
            Fault := #Fault,
            SecPulse := #SecPulse,
            AlwaysTrue := #AlwaysTrue,
            StartConfirmationPopupSel := 1,
            EndConfirmationPopupSel := #EndConfirmationPopupSel,
            WeightBasedSel := #WeightBasedSel,
            RMTypeSel := #RMTypeSel,
            AdditionMethodSel := #AdditionMethodSel,
            RMAddPopupSel := #RMAddPopupSel,
            "SetVacuum/SetPressure" := #"SetVacuum/SetPressure",
            SetQuantity := #SetQuantity,
            "ActualVacuum/ActualPressure" := #"ActualVacuum/ActualPressure",
            ActualQuantity := #ActualQuantity,
            ActualQuantityRMVessel := #ActualQuantityRMVessel,
            "VacuumTol/PressureTol" := #"VacuumTol/PressureTol",
            DelaytoSettleMaterial := #DelaytoSettleMaterial,
            InflightQuantity := #InflightQuantitySuction,
            SetRmNo := #SetRMNo,
            Start := #Start,
            Stop := #Stop,
            Reset := #Reset,
            StartConfirmationAck := #StartConfirmationAck,
            VacuumInValve => #VacuumInValve,
            VacuumLineValves => #VacuumLineValves,
            SuctionInValve => #SuctionInValve,
            VacuumPumpCmd => #VacuumPumpCmd,
            StartConfirmationPopup => #StartConfirmationPopup);
END_REGION

REGION Network 6: RM Addition Liquid Drum
